// SIMATIC S7-200 project (STEP 7-Micro/WIN), CPU 224 UN REL 02.01

SYMBOL_TABLE 01
数据记录             M0.0     // 0记录 1 不记录
光源模式             M0.1     // 光源模式切换 0新光源 1老光源
设置时钟B            M0.2     // 设置时钟按钮
间隔               M0.3
间隔使能             M0.4
整点               M0.5
在线               M0.6
离线               M0.7
报警复位             M1.0
维护               M1.1
启动标定             M1.2
启动测量             M1.3
自动标定             M1.4
恢复默认             M1.5
无源启动             M1.6
急停               M1.7
运行中              M2.0
实样标记             M3.3
启动质控             M3.4
质控标记             M3.5
质控标定标记           M3.7
量程切换开关           M4.0
加热开关             M5.1
负值显示             M5.2
正常结束             M11.0
连续测试状态           M11.2
历史使能             M20.0
empty            M23.0
进样标记             V19.0
标定中              V20.0
标定阶段0            V20.1
标定阶段1            V20.4
标定阶段2            V21.0
测量中              V22.0
第一档              V91.0
第二档              V91.1
第三档              V91.2
第四档              V91.3
第五档              V91.4
档位               VB90     // 0：第一档  1：第二档  2：第三档  3：第四档
切换范围             VB92
自标时              VB258
自标分              VB259
时钟字节             VB400    // BCD
时钟时              VB403
时钟分              VB404
显色               VD220
基准               VD224
校正系数             VD270
负值区间             VD274
操作密码             VD306
管理密码             VD310
超级密码             VD314
中间值              VD490
模拟输出             VD494
平均电压             VD582
临时A0             VD636
平均A0             VD640
平均A1             VD644
平均A2             VD648
临时A1             VD656
临时A2             VD660
仪器动作             VW94
仪器状态             VW96
占空比              VW218
间隔时              VW230
间隔分              VW232
质不过              VW260
质已测              VW262
切换次数             VW264
标0次数             VW326
标1次数             VW328
标2次数             VW330
HMI窗口号           VW390
时钟字              VW410    // BCD
测量启动时间           VW450
断电时刻             VW470
END_SYMBOL_TABLE

SYMBOL_TABLE 输入输出
下三通信号            I0.0
上三通信号            I0.1
水样浮球             I1.2
废液浮球             I1.3
加热               Q0.0
光源               Q0.1
加热保护             Q0.2
END_SYMBOL_TABLE

SYMBOL_TABLE 自动
A试剂a             V0.0     // 重铬酸钾
B试剂a             V0.1
C试剂a             V0.2     // 硫酸
D试剂a             V0.3
X试剂a             V0.4
纯水a              V0.5
清洗液a             V0.6
水样a              V0.7
空气a              V1.0
进样阀a             V1.1
切水样阀a            V1.2
高压阀a             V1.3
上摇臂a             V1.4
下摇臂a             V1.5
P1抽a             V1.6
P1推a             V1.7
P2抽a             V2.0
P2推a             V2.1
P外a              V2.2
风扇a              V2.3
校一a              V2.4
校二a              V2.5
光源a              V2.6
样校水              V2.7
采样球阀a            V3.0     // 常闭
排空球阀2a           V3.1     // 常开
硫酸a              V3.2
重铬酸钾a            V3.3
备用1a             V3.4
END_SYMBOL_TABLE

SYMBOL_TABLE 参数
校一浓度             VD100    // 浮
校二浓度             VD104    // 浮
消解时间             VW108    // min
显色时间             VW110    // min
采样报警时间           VW112    // min
罐溢流时间            VW114    // s
管溢流时间            VW116    // s
                 VW118    // 测量模式
                 VW120    // 自动标定启用
自标周期             VW122    // 天
当前计算             VW124    // 天
模拟量程             VD126    // mg/L   浮
消解温度             VD130    // 浮
版本号              VD134    // 浮
启动时刻             VW138    // hex   ,vw134-vw142
标定时刻             VW148    // hex    ,vw144-152
K                VD158    // 浮
B                VD162    // 浮
水样A              VD166    // 浮
水样T              VD170    // 浮
校正液T             VD174    // 浮
纯水T              VD178    // 浮
校一A              VD182    // 浮
校二A              VD186    // 浮
当前温度             VD190    // 浮
当前电压             VD194    // 浮
排空电压             VD1100
清洗电压             VD1104
目标温度             VD200
显色温度             VD204
END_SYMBOL_TABLE

SYMBOL_TABLE 报警
A试剂报警            V80.0    // Vb80-81二级报警 ,停止一切操作
B试剂报警            V80.1
C试剂报警            V80.2
D试剂报警            V80.3
X试剂报警            V80.4
纯水报警             V80.5
硫酸报警             V80.6
废液满              V81.0
校一报警             V81.1
校二报警             V81.2
采样报警             V82.1
重铬酸钾报警           V81.4
清洗液报警            V81.5
在线样报警            V82.0    // vb82一级报警，自动测量不停
消解温度异常           V83.0
待机温度异常           V83.1
冷却超时             V83.2
基准偏低             V83.3
END_SYMBOL_TABLE

SYMBOL_TABLE S7-200 符号
Always_On        SM0.0    // 始终接通为 ON
First_Scan_On    SM0.1    // 仅第一个扫描周期中接通为 ON
Clock_1s         SM0.5    // 在 1 秒钟的循环周期内，接通为 ON 0.5 秒，关断为 OFF 0.5  秒
END_SYMBOL_TABLE

ORGANIZATION_BLOCK 程序块:OB1
TITLE=
BEGIN
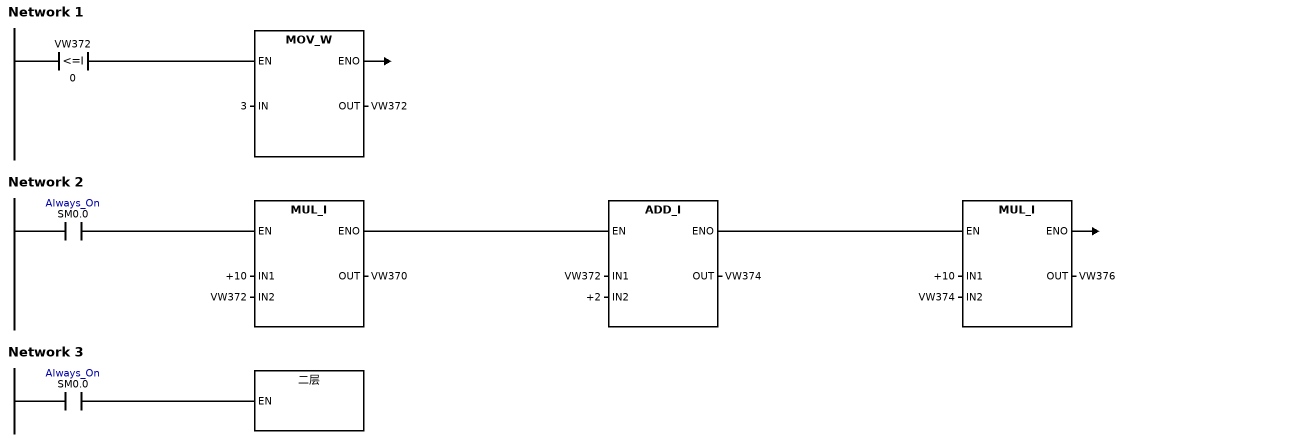
Network 1
LDW<=  VW372, 0
MOVW   3, VW372
Network 2
LD     Always_On:SM0.0
MOVW   +10, VW370
AENO
*I     VW372, VW370
AENO
MOVW   VW372, VW374
AENO
+I     +2, VW374
AENO
MOVW   +10, VW376
*I     VW374, VW376
Network 3
LD     Always_On:SM0.0
CALL   二层:SBR10
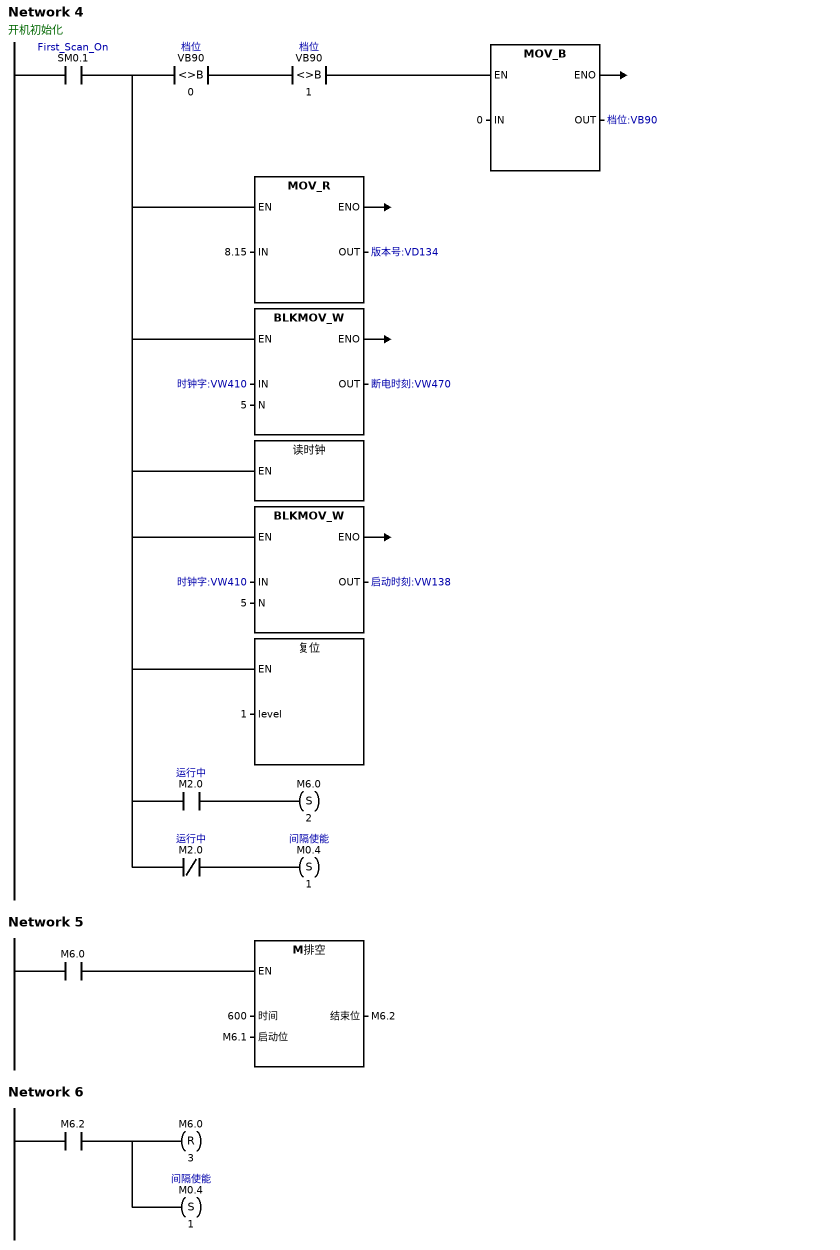
Network 4
// 开机初始化
LD     First_Scan_On:SM0.1
LPS
AB<>   档位:VB90, 0
AB<>   档位:VB90, 1
MOVB   0, 档位:VB90
LRD
MOVR   8.15, 版本号:VD134
LRD
BMW    时钟字:VW410, 断电时刻:VW470, 5
LRD
CALL   读时钟:SBR28
LRD
BMW    时钟字:VW410, 启动时刻:VW138, 5
LRD
CALL   复位:SBR34, 1
LRD
A      运行中:M2.0
S      M6.0, 2
LPP
AN     运行中:M2.0
S      间隔使能:M0.4, 1
Network 5
LD     M6.0
CALL   M排空:SBR5, 600, M6.1, M6.2
Network 6
LD     M6.2
R      M6.0, 3
S      间隔使能:M0.4, 1
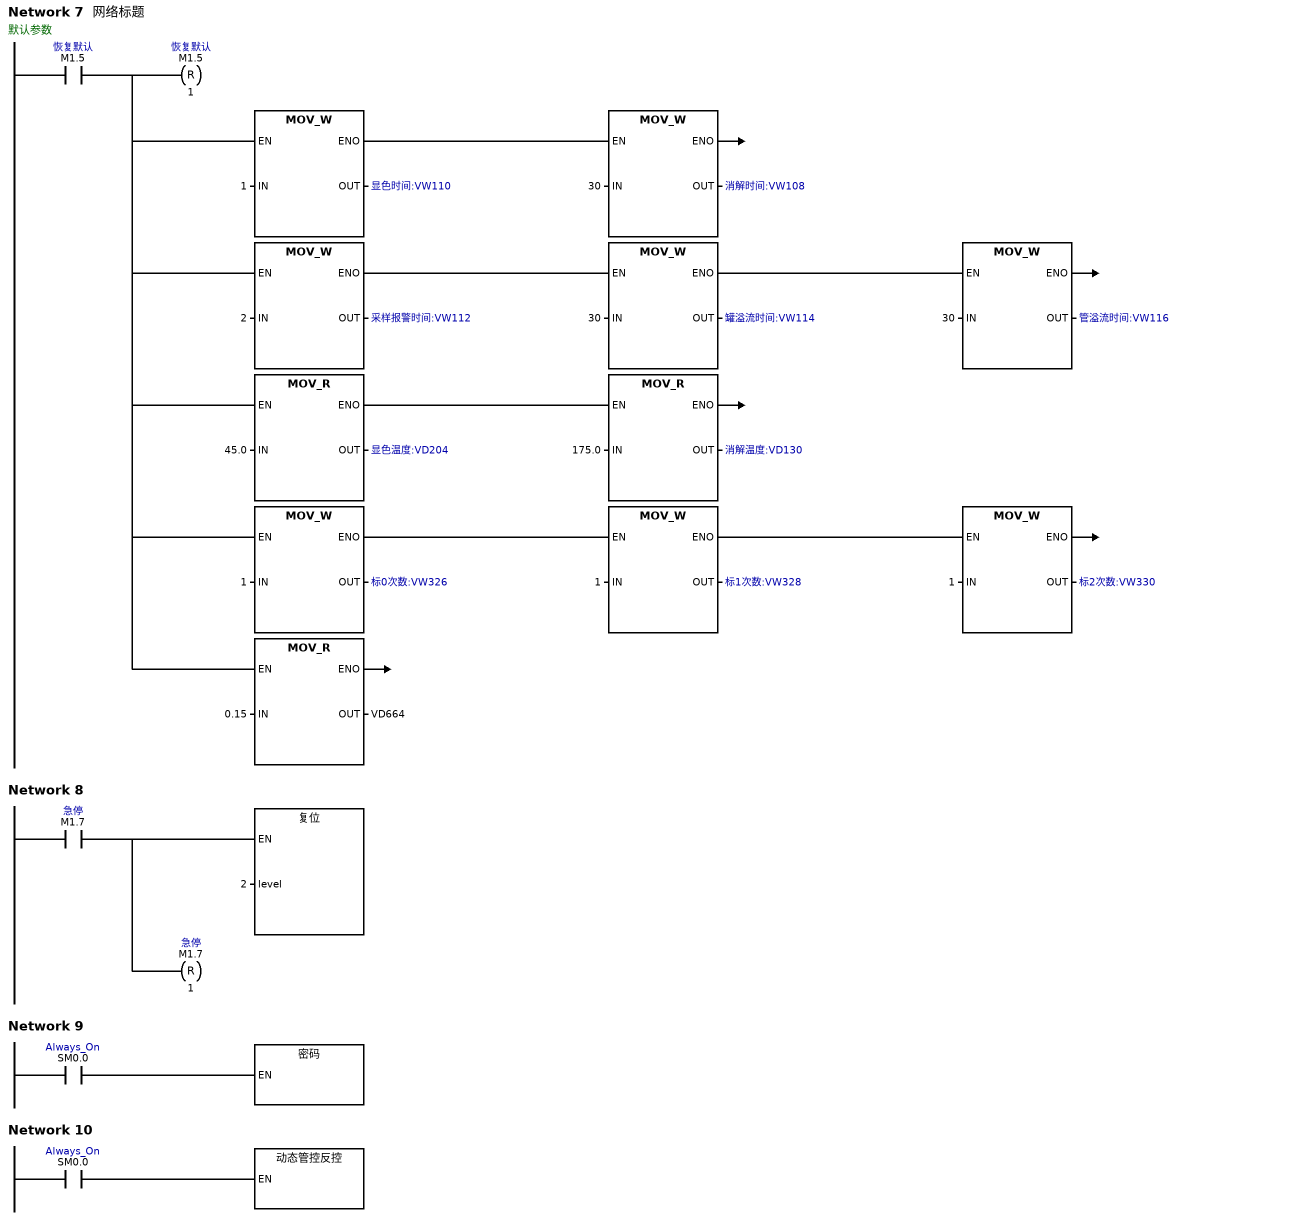
Network 7 // 网络标题
// 默认参数
LD     恢复默认:M1.5
LPS
R      恢复默认:M1.5, 1
MOVW   1, 显色时间:VW110
AENO
MOVW   30, 消解时间:VW108
LRD
MOVW   2, 采样报警时间:VW112
AENO
MOVW   30, 罐溢流时间:VW114
AENO
MOVW   30, 管溢流时间:VW116
LRD
MOVR   45.0, 显色温度:VD204
AENO
MOVR   175.0, 消解温度:VD130
LRD
MOVW   1, 标0次数:VW326
AENO
MOVW   1, 标1次数:VW328
AENO
MOVW   1, 标2次数:VW330
LPP
MOVR   0.15, VD664
Network 8
LD     急停:M1.7
CALL   复位:SBR34, 2
R      急停:M1.7, 1
Network 9
LD     Always_On:SM0.0
CALL   密码:SBR26
Network 10
LD     Always_On:SM0.0
CALL   动态管控反控:SBR38
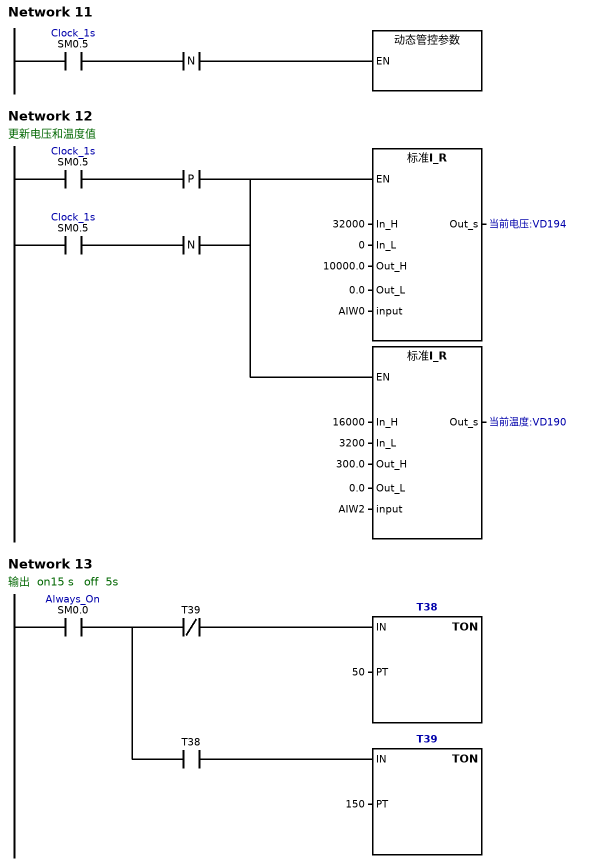
Network 11
LD     Clock_1s:SM0.5
ED
CALL   动态管控参数:SBR24
Network 12
// 更新电压和温度值
LD     Clock_1s:SM0.5
EU
LD     Clock_1s:SM0.5
ED
OLD
CALL   标准I_R:SBR2, 32000, 0, 10000.0, 0.0, AIW0, 当前电压:VD194
CALL   标准I_R:SBR2, 16000, 3200, 300.0, 0.0, AIW2, 当前温度:VD190
Network 13
// 输出  on15 s   off  5s
LD     Always_On:SM0.0
LPS
AN     T39
TON    T38, 50
LPP
A      T38
TON    T39, 150
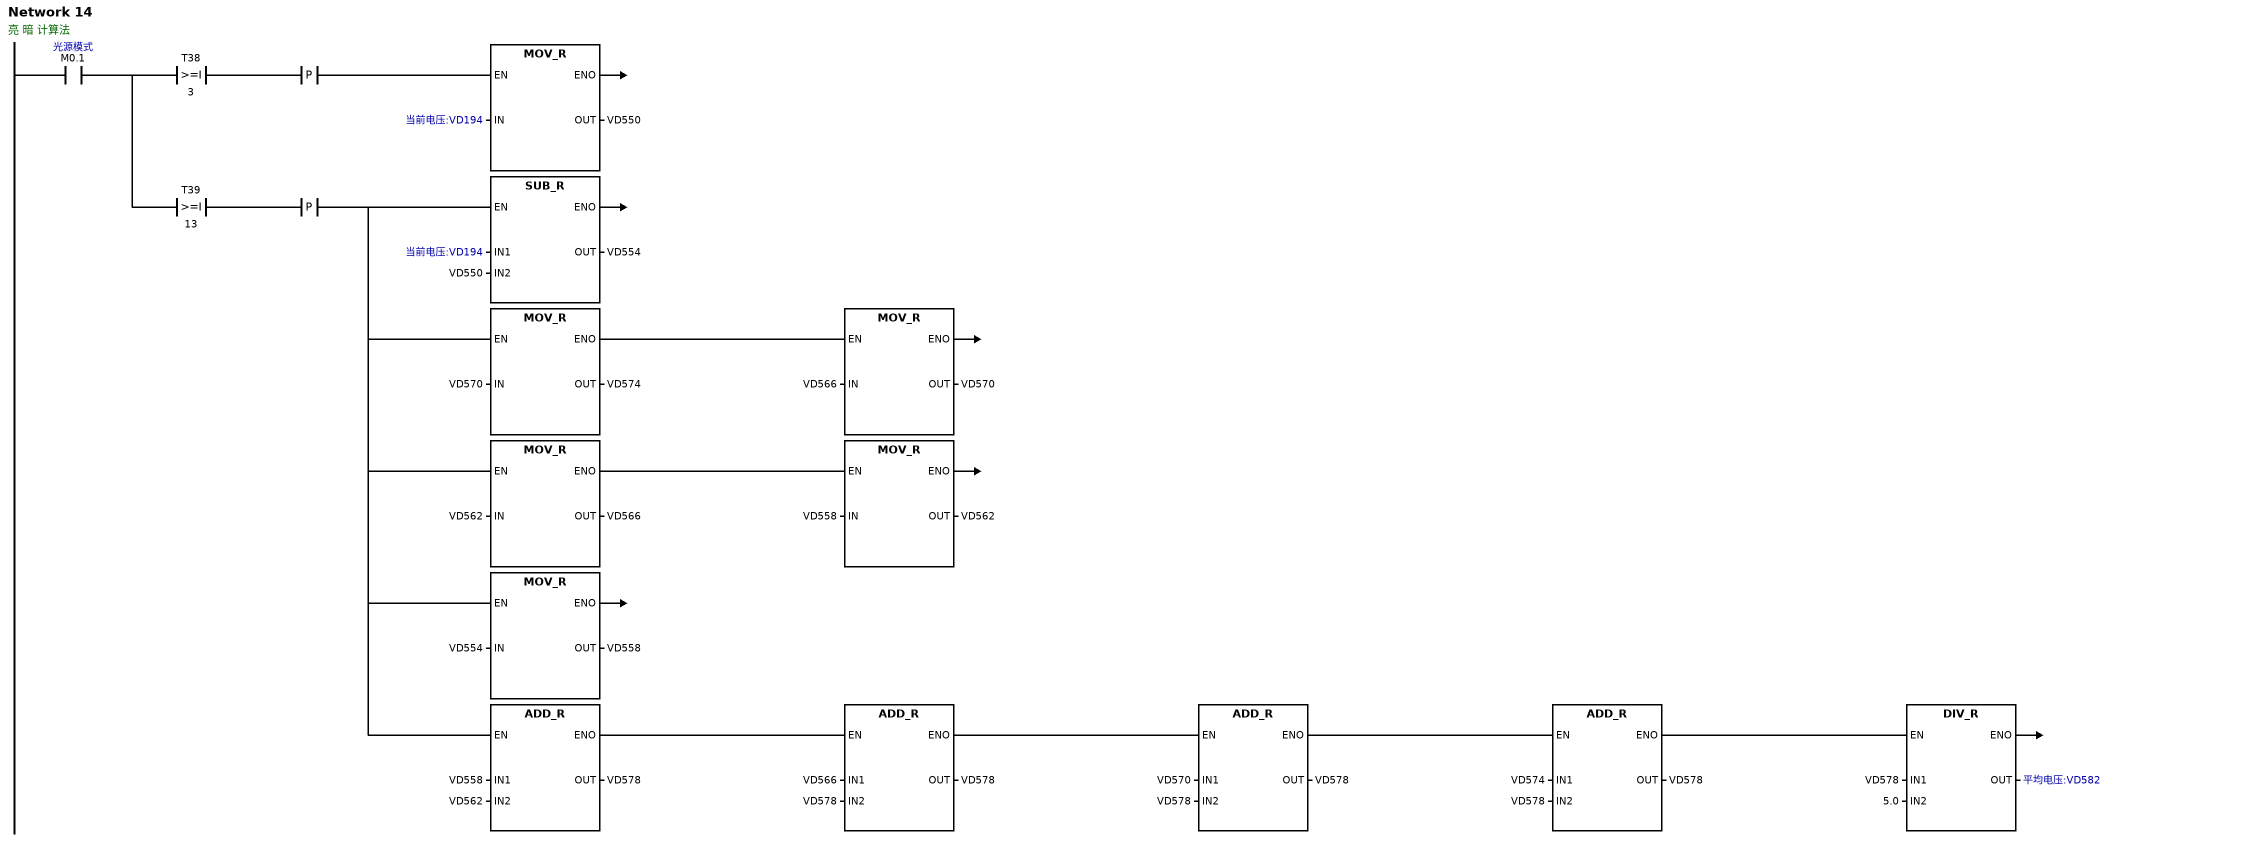
Network 14
// 亮 暗 计算法
LD     光源模式:M0.1
LPS
AW>=   T38, 3
EU
MOVR   当前电压:VD194, VD550
LPP
AW>=   T39, 13
EU
LPS
MOVR   当前电压:VD194, VD554
-R     VD550, VD554
MOVR   VD570, VD574
AENO
MOVR   VD566, VD570
LRD
MOVR   VD562, VD566
AENO
MOVR   VD558, VD562
LRD
MOVR   VD554, VD558
LPP
MOVR   VD558, VD578
AENO
+R     VD562, VD578
AENO
+R     VD566, VD578
AENO
+R     VD570, VD578
AENO
+R     VD574, VD578
AENO
MOVR   VD578, 平均电压:VD582
/R     5.0, 平均电压:VD582
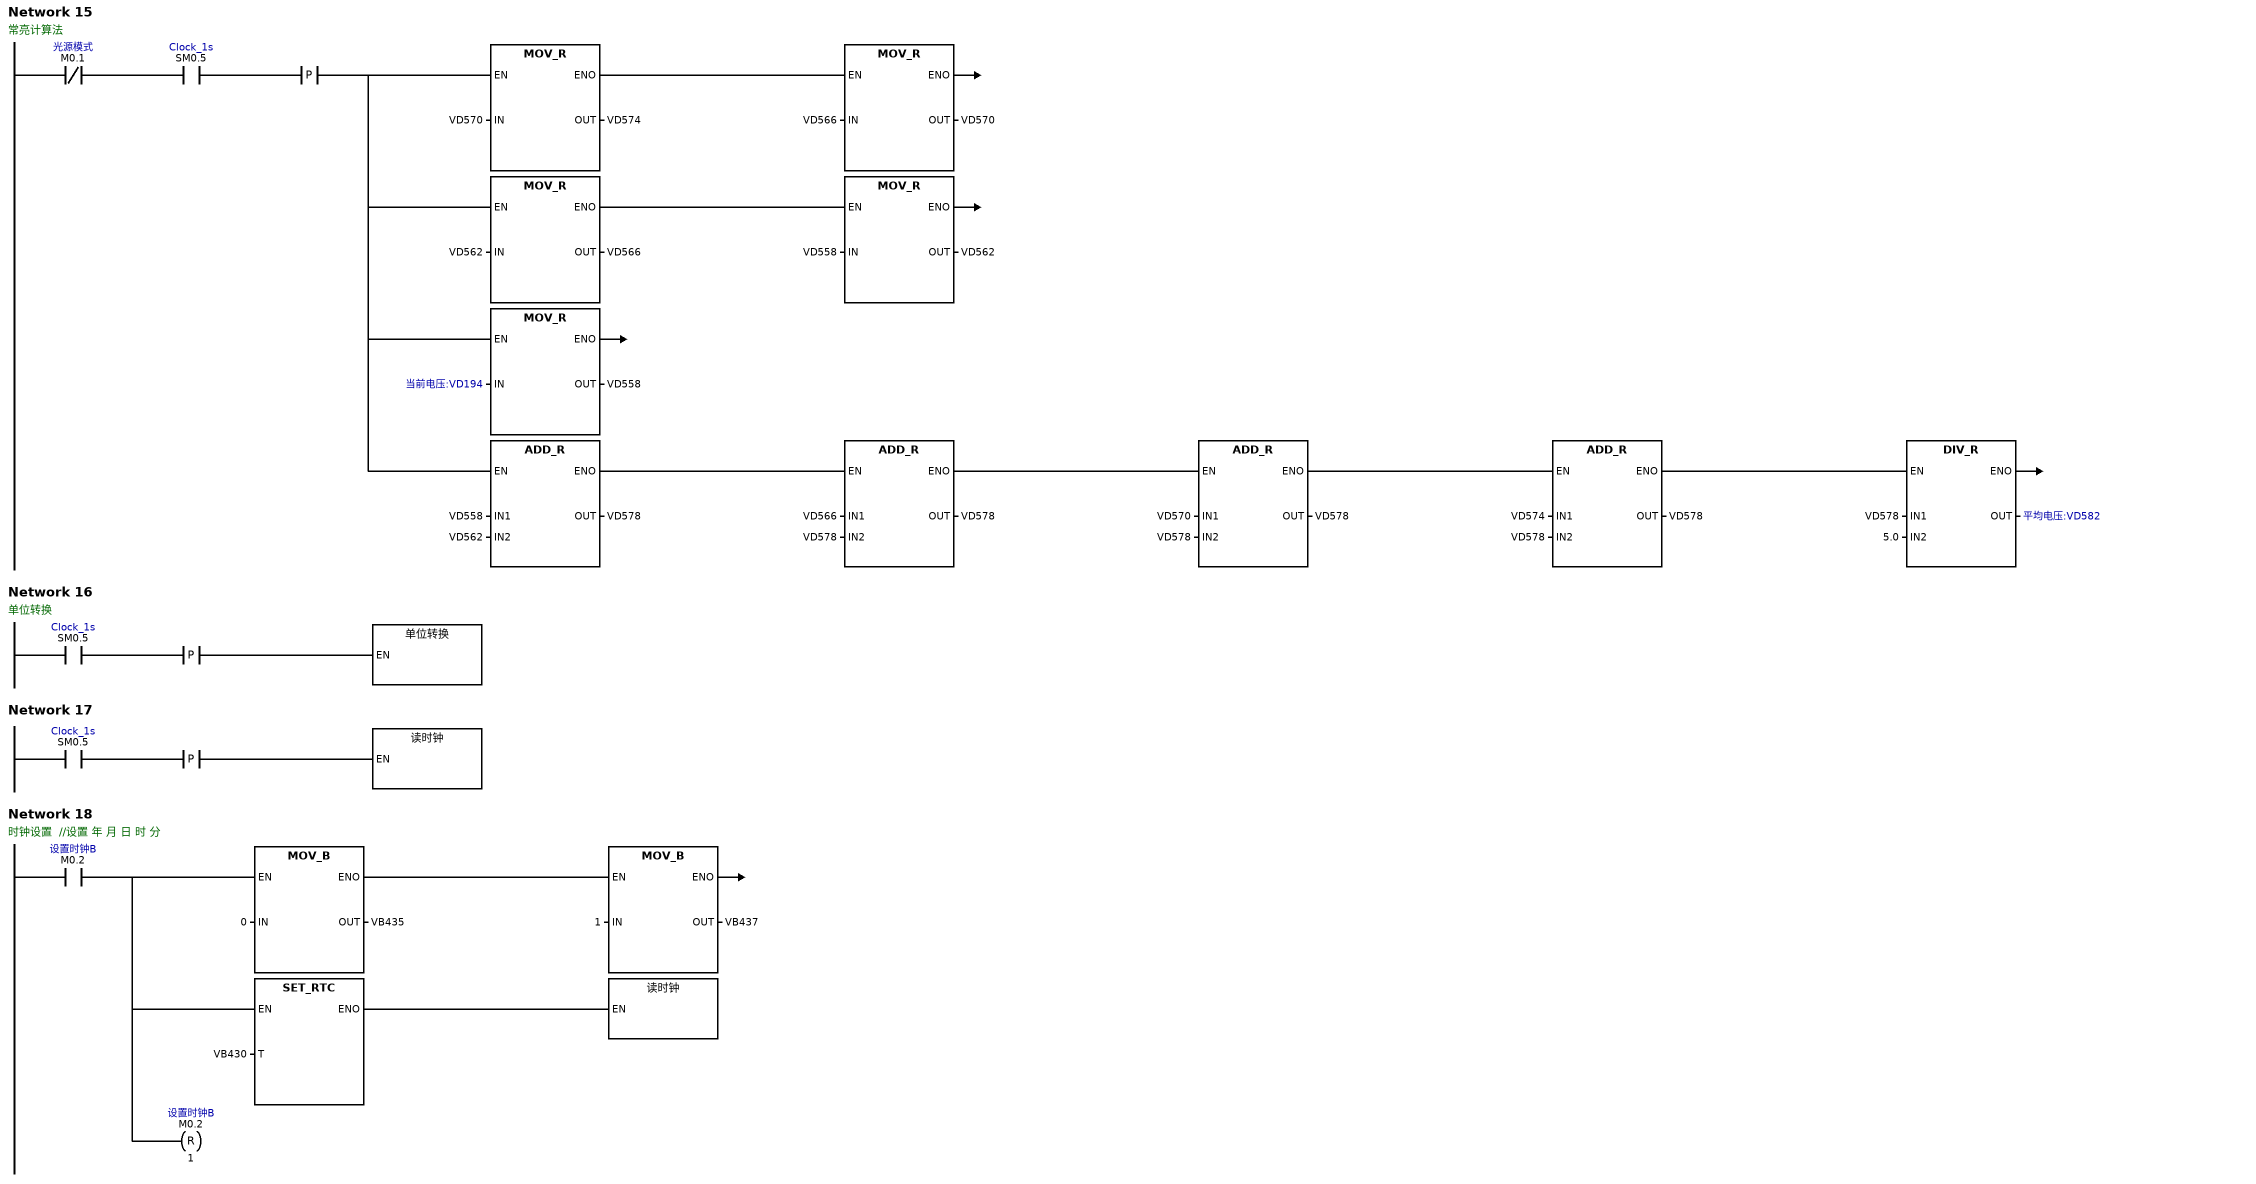
Network 15
// 常亮计算法
LDN    光源模式:M0.1
A      Clock_1s:SM0.5
EU
LPS
MOVR   VD570, VD574
AENO
MOVR   VD566, VD570
LRD
MOVR   VD562, VD566
AENO
MOVR   VD558, VD562
LRD
MOVR   当前电压:VD194, VD558
LPP
MOVR   VD558, VD578
AENO
+R     VD562, VD578
AENO
+R     VD566, VD578
AENO
+R     VD570, VD578
AENO
+R     VD574, VD578
AENO
MOVR   VD578, 平均电压:VD582
/R     5.0, 平均电压:VD582
Network 16
// 单位转换
LD     Clock_1s:SM0.5
EU
CALL   单位转换:SBR27
Network 17
LD     Clock_1s:SM0.5
EU
CALL   读时钟:SBR28
Network 18
// 时钟设置  //设置 年 月 日 时 分
LD     设置时钟B:M0.2
LPS
MOVB   0, VB435
AENO
MOVB   1, VB437
LRD
TODW   VB430
AENO
CALL   读时钟:SBR28
LPP
R      设置时钟B:M0.2, 1
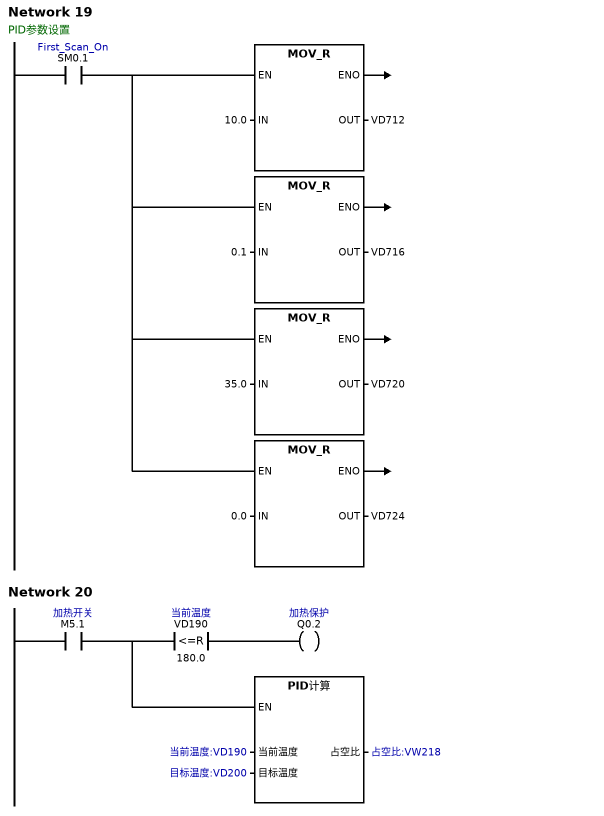
Network 19
// PID参数设置
LD     First_Scan_On:SM0.1
MOVR   10.0, VD712
MOVR   0.1, VD716
MOVR   35.0, VD720
MOVR   0.0, VD724
Network 20
LD     加热开关:M5.1
LPS
AR<=   当前温度:VD190, 180.0
=      加热保护:Q0.2
LPP
CALL   PID计算:SBR9, 当前温度:VD190, 目标温度:VD200, 占空比:VW218
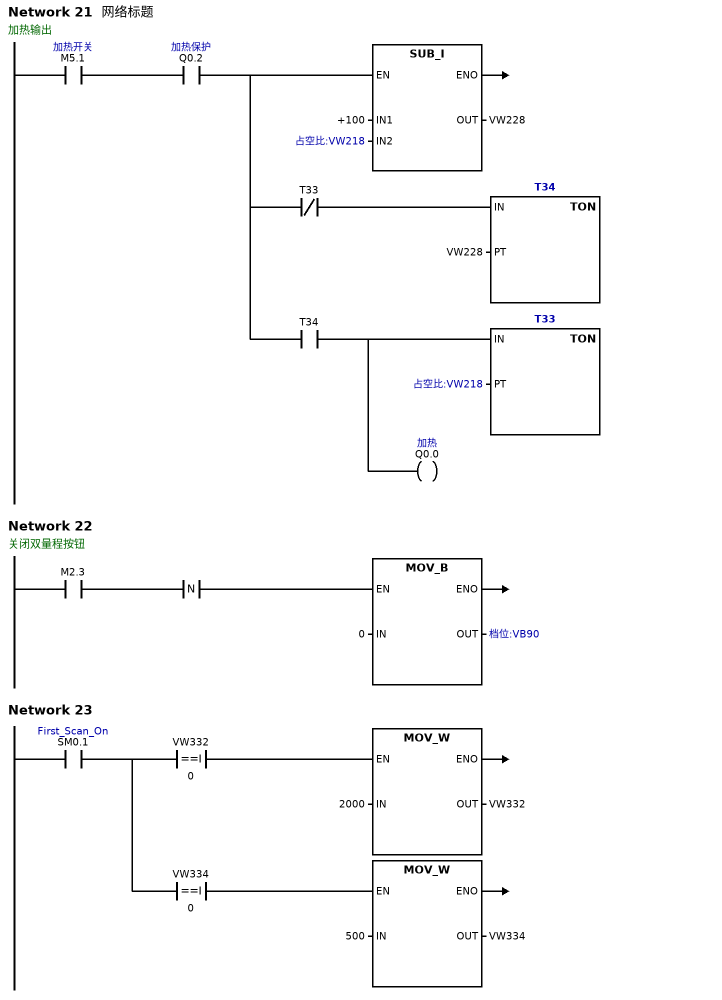
Network 21 // 网络标题
//   加热输出
LD     加热开关:M5.1
A      加热保护:Q0.2
LPS
MOVW   +100, VW228
-I     占空比:VW218, VW228
AN     T33
TON    T34, VW228
LPP
A      T34
TON    T33, 占空比:VW218
=      加热:Q0.0
Network 22
// 关闭双量程按钮
LD     M2.3
ED
MOVB   0, 档位:VB90
Network 23
LD     First_Scan_On:SM0.1
LPS
AW=    VW332, 0
MOVW   2000, VW332
LPP
AW=    VW334, 0
MOVW   500, VW334
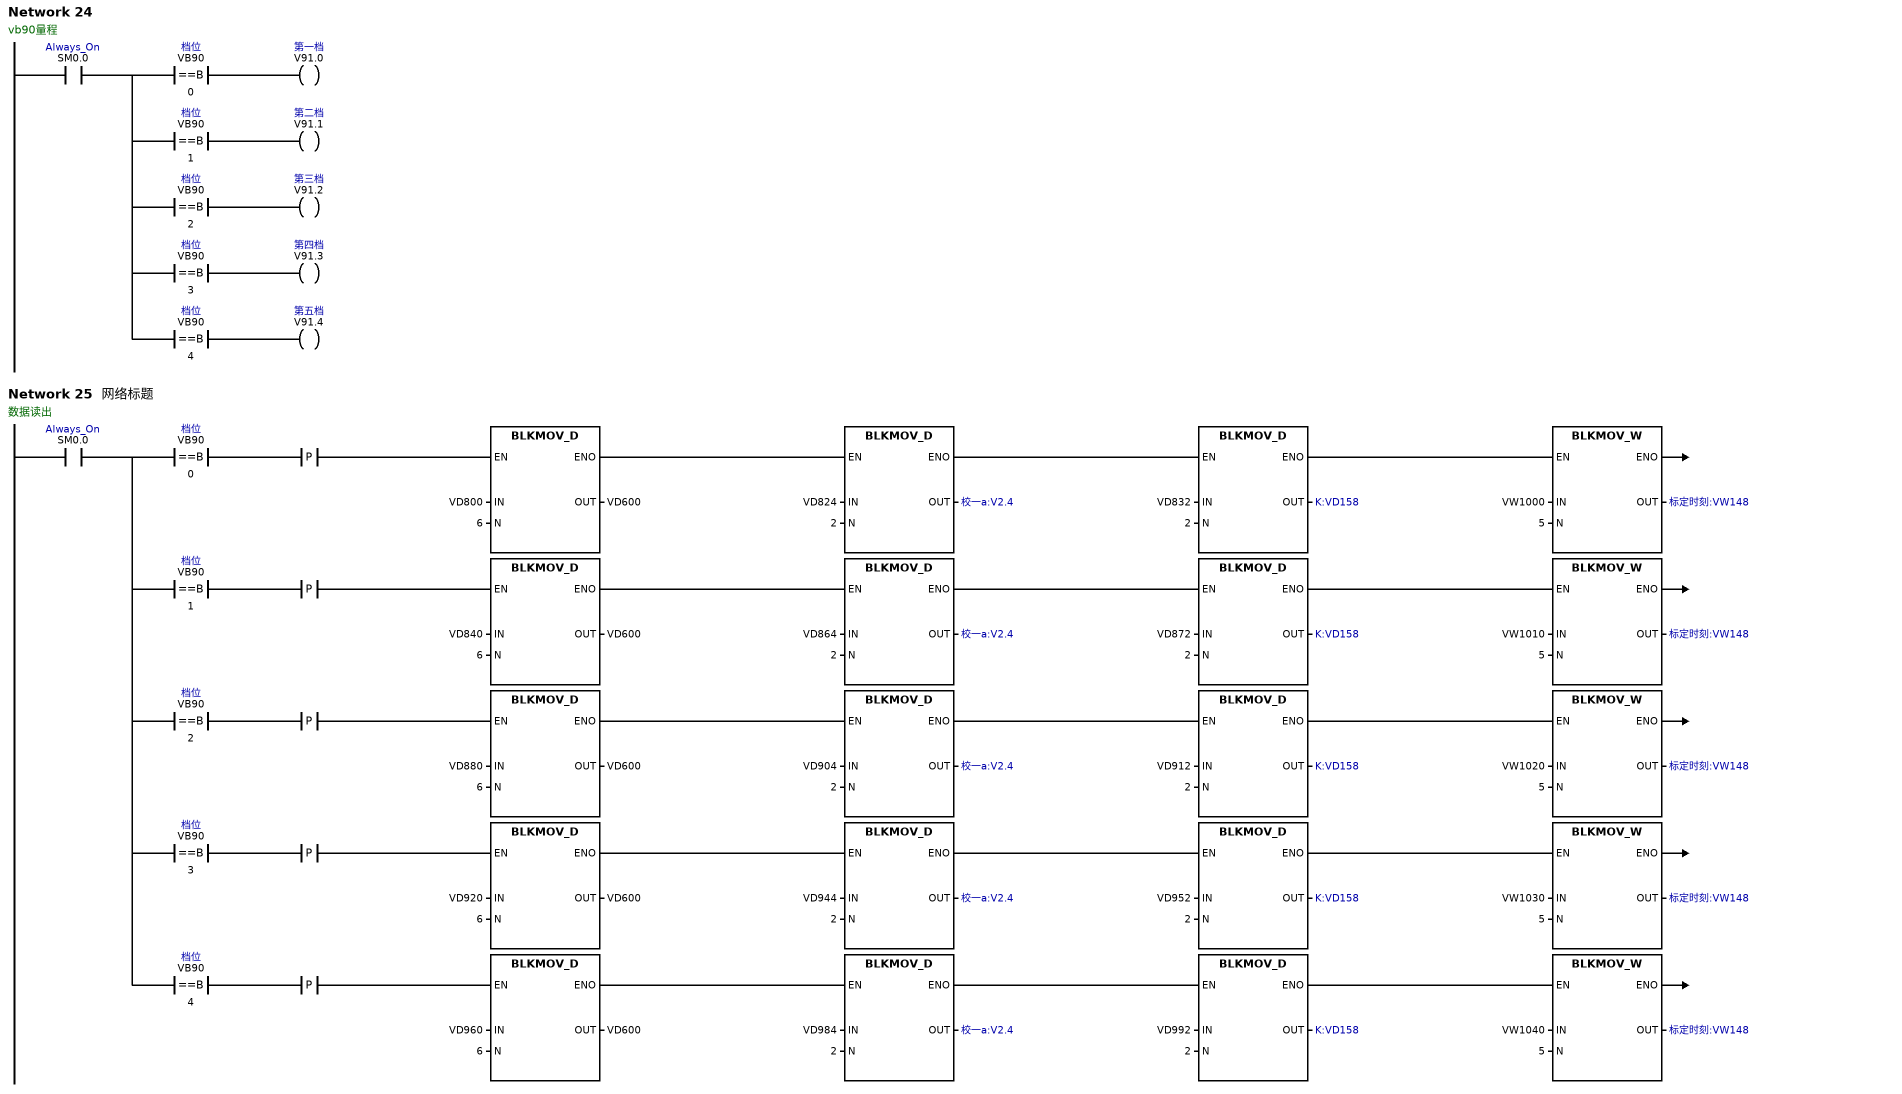
Network 24
// vb90量程
LD     Always_On:SM0.0
LPS
AB=    档位:VB90, 0
=      第一档:V91.0
LRD
AB=    档位:VB90, 1
=      第二档:V91.1
LRD
AB=    档位:VB90, 2
=      第三档:V91.2
LRD
AB=    档位:VB90, 3
=      第四档:V91.3
LPP
AB=    档位:VB90, 4
=      第五档:V91.4
Network 25 // 网络标题
// 数据读出
// (network saved uncompiled; LAD cells follow)
// row 0: c0 -| |- Always_On:SM0.0 v  c1 -|==B|- 档位:VB90, 0  c2 -|P|-  c3 --  c4 [BLKMOV_D EN:=power@row0, IN:=VD800, N:=6, ENO=>power, OUT=>VD600]  c5 --  c6 --  c7 [BLKMOV_D EN:=power@row0, IN:=VD824, N:=2, ENO=>power, OUT=>校一a:V2.4]  c8 --  c9 --  c10 [BLKMOV_D EN:=power@row0, IN:=VD832, N:=2, ENO=>power, OUT=>K:VD158]  c11 --  c12 --  c13 [BLKMOV_W EN:=power@row0, IN:=VW1000, N:=5, ENO=>power, OUT=>标定时刻:VW148]  c14 ->
// row 1: c0 ^v  c4 [box]  c7 [box]  c10 [box]  c13 [box]
// row 2: c0 ^v  c1 -|==B|- 档位:VB90, 1  c2 -|P|-  c3 --  c4 [BLKMOV_D EN:=power@row2, IN:=VD840, N:=6, ENO=>power, OUT=>VD600]  c5 --  c6 --  c7 [BLKMOV_D EN:=power@row2, IN:=VD864, N:=2, ENO=>power, OUT=>校一a:V2.4]  c8 --  c9 --  c10 [BLKMOV_D EN:=power@row2, IN:=VD872, N:=2, ENO=>power, OUT=>K:VD158]  c11 --  c12 --  c13 [BLKMOV_W EN:=power@row2, IN:=VW1010, N:=5, ENO=>power, OUT=>标定时刻:VW148]  c14 ->
// row 3: c0 ^v  c4 [box]  c7 [box]  c10 [box]  c13 [box]
// row 4: c0 ^v  c1 -|==B|- 档位:VB90, 2  c2 -|P|-  c3 --  c4 [BLKMOV_D EN:=power@row4, IN:=VD880, N:=6, ENO=>power, OUT=>VD600]  c5 --  c6 --  c7 [BLKMOV_D EN:=power@row4, IN:=VD904, N:=2, ENO=>power, OUT=>校一a:V2.4]  c8 --  c9 --  c10 [BLKMOV_D EN:=power@row4, IN:=VD912, N:=2, ENO=>power, OUT=>K:VD158]  c11 --  c12 --  c13 [BLKMOV_W EN:=power@row4, IN:=VW1020, N:=5, ENO=>power, OUT=>标定时刻:VW148]  c14 ->
// row 5: c0 ^v  c4 [box]  c7 [box]  c10 [box]  c13 [box]
// row 6: c0 ^v  c1 -|==B|- 档位:VB90, 3  c2 -|P|-  c3 --  c4 [BLKMOV_D EN:=power@row6, IN:=VD920, N:=6, ENO=>power, OUT=>VD600]  c5 --  c6 --  c7 [BLKMOV_D EN:=power@row6, IN:=VD944, N:=2, ENO=>power, OUT=>校一a:V2.4]  c8 --  c9 --  c10 [BLKMOV_D EN:=power@row6, IN:=VD952, N:=2, ENO=>power, OUT=>K:VD158]  c11 --  c12 --  c13 [BLKMOV_W EN:=power@row6, IN:=VW1030, N:=5, ENO=>power, OUT=>标定时刻:VW148]  c14 ->
// row 7: c0 ^v  c4 [box]  c7 [box]  c10 [box]  c13 [box]
// row 8: c0 ^  c1 -|==B|- 档位:VB90, 4  c2 -|P|-  c3 --  c4 [BLKMOV_D EN:=power@row8, IN:=VD960, N:=6, ENO=>power, OUT=>VD600]  c5 --  c6 --  c7 [BLKMOV_D EN:=power@row8, IN:=VD984, N:=2, ENO=>power, OUT=>校一a:V2.4]  c8 --  c9 --  c10 [BLKMOV_D EN:=power@row8, IN:=VD992, N:=2, ENO=>power, OUT=>K:VD158]  c11 --  c12 --  c13 [BLKMOV_W EN:=power@row8, IN:=VW1040, N:=5, ENO=>power, OUT=>标定时刻:VW148]  c14 ->
// row 9: c4 [box]  c7 [box]  c10 [box]  c13 [box]
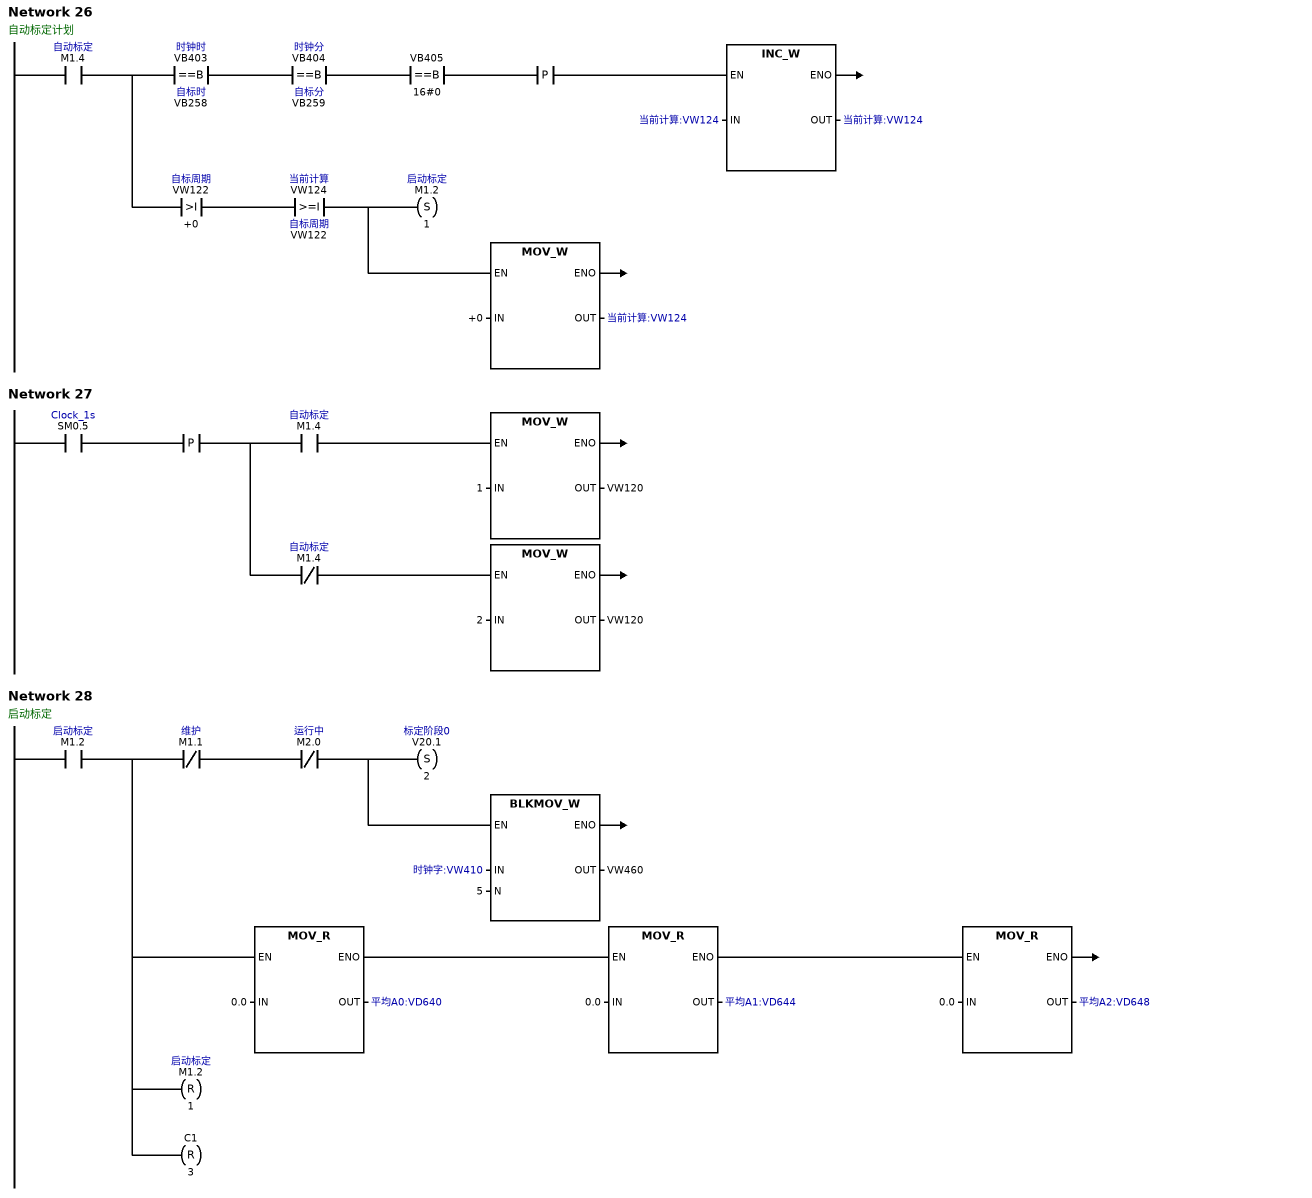
Network 26
// 自动标定计划
LD     自动标定:M1.4
LPS
AB=    时钟时:VB403, 自标时:VB258
AB=    时钟分:VB404, 自标分:VB259
AB=    VB405, 16#0
EU
INCW   当前计算:VW124
LPP
AW>    自标周期:VW122, +0
AW>=   当前计算:VW124, 自标周期:VW122
S      启动标定:M1.2, 1
MOVW   +0, 当前计算:VW124
Network 27
LD     Clock_1s:SM0.5
EU
LPS
A      自动标定:M1.4
MOVW   1, VW120
LPP
AN     自动标定:M1.4
MOVW   2, VW120
Network 28
// 启动标定
LD     启动标定:M1.2
LPS
AN     维护:M1.1
AN     运行中:M2.0
S      标定阶段0:V20.1, 2
BMW    时钟字:VW410, VW460, 5
LPP
LPS
MOVR   0.0, 平均A0:VD640
AENO
MOVR   0.0, 平均A1:VD644
AENO
MOVR   0.0, 平均A2:VD648
LRD
R      启动标定:M1.2, 1
LPP
R      C1, 3
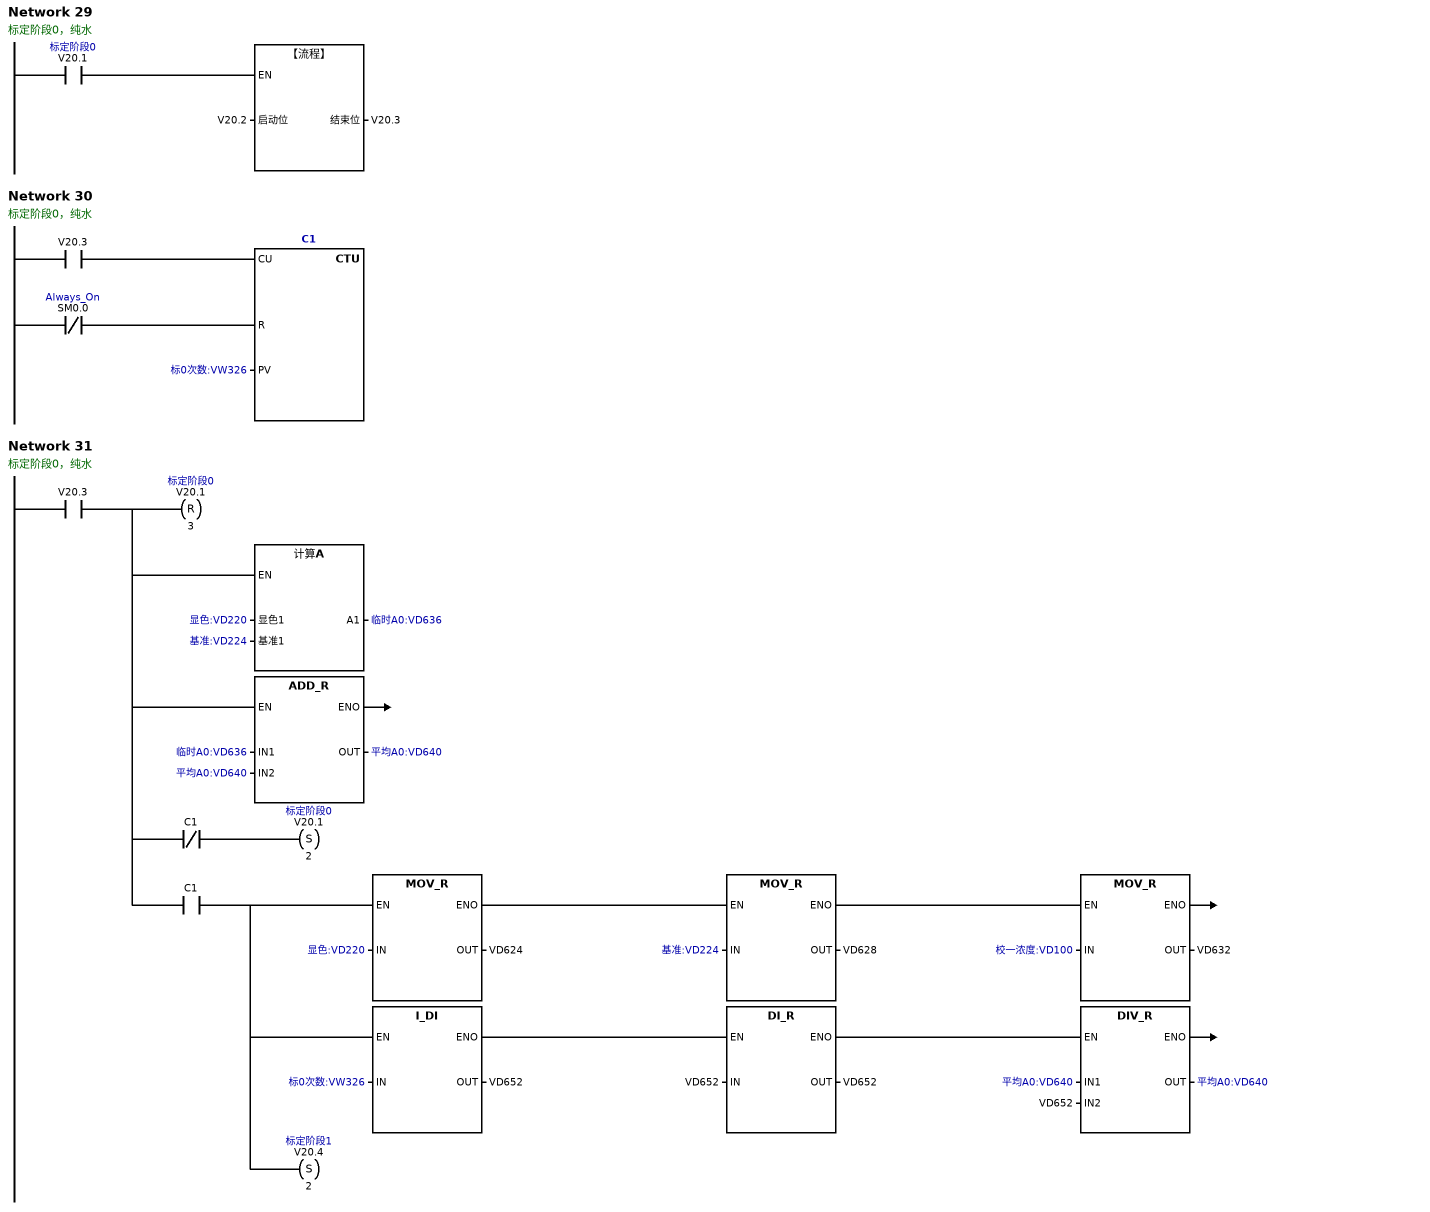
Network 29
// 标定阶段0，纯水
LD     标定阶段0:V20.1
CALL   【流程】:SBR7, V20.2, V20.3
Network 30
// 标定阶段0，纯水
LD     V20.3
LDN    Always_On:SM0.0
CTU    C1, 标0次数:VW326
Network 31
// 标定阶段0，纯水
LD     V20.3
LPS
R      标定阶段0:V20.1, 3
CALL   计算A:SBR37, 显色:VD220, 基准:VD224, 临时A0:VD636
+R     临时A0:VD636, 平均A0:VD640
AN     C1
S      标定阶段0:V20.1, 2
LPP
A      C1
LPS
MOVR   显色:VD220, VD624
AENO
MOVR   基准:VD224, VD628
AENO
MOVR   校一浓度:VD100, VD632
LRD
ITD    标0次数:VW326, VD652
AENO
DTR    VD652, VD652
AENO
/R     VD652, 平均A0:VD640
LPP
S      标定阶段1:V20.4, 2
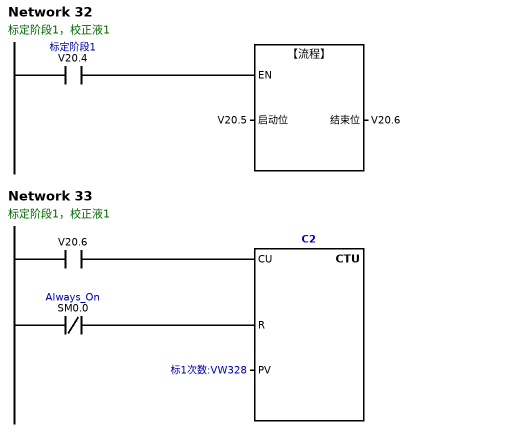
Network 32
// 标定阶段1，校正液1
LD     标定阶段1:V20.4
CALL   【流程】:SBR7, V20.5, V20.6
Network 33
// 标定阶段1，校正液1
LD     V20.6
LDN    Always_On:SM0.0
CTU    C2, 标1次数:VW328
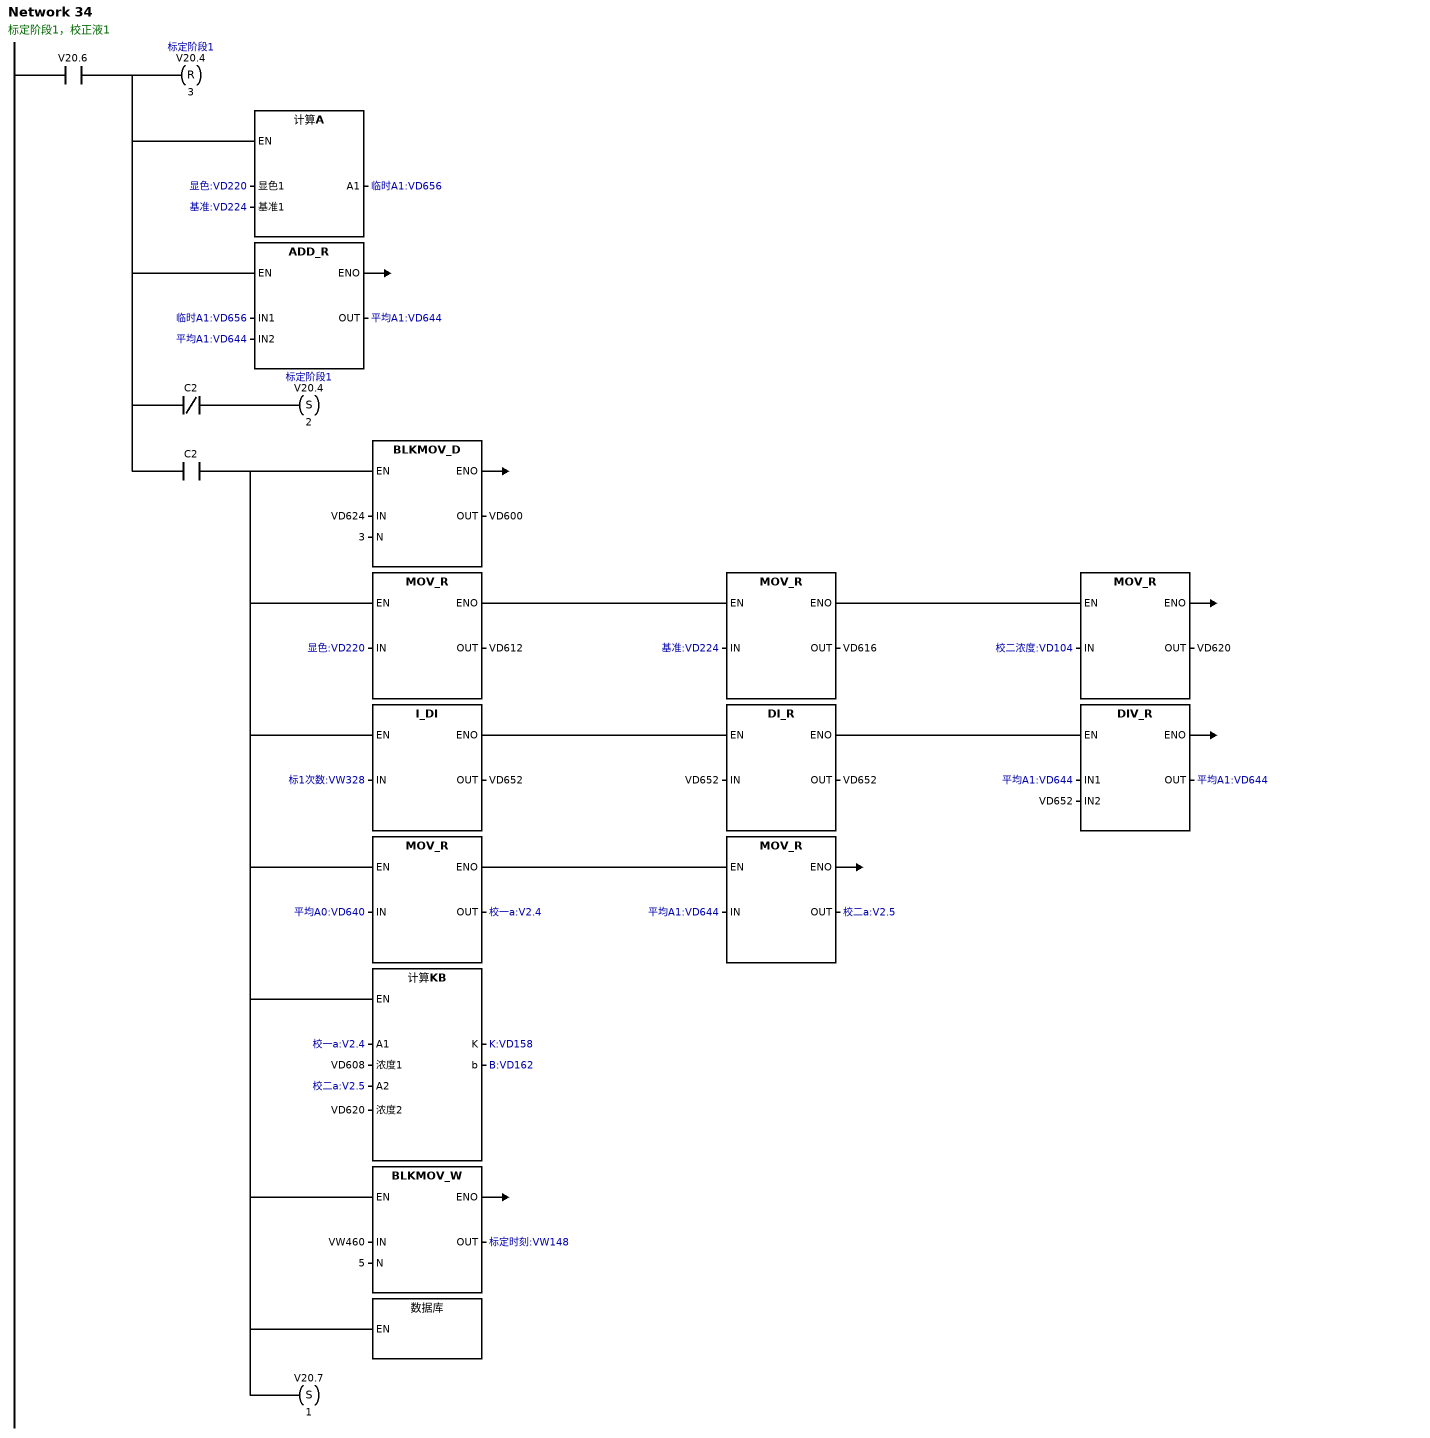
Network 34
// 标定阶段1，校正液1
// (network saved uncompiled; LAD cells follow)
// row 0: c0 -| |- V20.6 v  c1 -(R) 标定阶段1:V20.4, 3
// row 1: c0 ^v  c1 --  c2 [计算A EN:=power@row1, 显色1:=显色:VD220, 基准1:=基准:VD224, A1=>临时A1:VD656]
// row 2: c0 ^v  c2 [box]
// row 3: c0 ^v  c1 --  c2 [ADD_R EN:=power@row3, IN1:=临时A1:VD656, IN2:=平均A1:VD644, ENO=>power, OUT=>平均A1:VD644]  c3 ->
// row 4: c0 ^v  c2 [box]
// row 5: c0 ^v  c1 -|/|- C2  c2 -(S) 标定阶段1:V20.4, 2
// row 6: c0 ^  c1 -| |- C2 v  c2 --  c3 [BLKMOV_D EN:=power@row6, IN:=VD624, N:=3, ENO=>power, OUT=>VD600]  c4 ->
// row 7: c1 ^v  c3 [box]
// row 8: c1 ^v  c2 --  c3 [MOV_R EN:=power@row8, IN:=显色:VD220, ENO=>power, OUT=>VD612]  c4 --  c5 --  c6 [MOV_R EN:=power@row8, IN:=基准:VD224, ENO=>power, OUT=>VD616]  c7 --  c8 --  c9 [MOV_R EN:=power@row8, IN:=校二浓度:VD104, ENO=>power, OUT=>VD620]  c10 ->
// row 9: c1 ^v  c3 [box]  c6 [box]  c9 [box]
// row 10: c1 ^v  c2 --  c3 [I_DI EN:=power@row10, IN:=标1次数:VW328, ENO=>power, OUT=>VD652]  c4 --  c5 --  c6 [DI_R EN:=power@row10, IN:=VD652, ENO=>power, OUT=>VD652]  c7 --  c8 --  c9 [DIV_R EN:=power@row10, IN1:=平均A1:VD644, IN2:=VD652, ENO=>power, OUT=>平均A1:VD644]  c10 ->
// row 11: c1 ^v  c3 [box]  c6 [box]  c9 [box]
// row 12: c1 ^v  c2 --  c3 [MOV_R EN:=power@row12, IN:=平均A0:VD640, ENO=>power, OUT=>校一a:V2.4]  c4 --  c5 --  c6 [MOV_R EN:=power@row12, IN:=平均A1:VD644, ENO=>power, OUT=>校二a:V2.5]  c7 ->
// row 13: c1 ^v  c3 [box]  c6 [box]
// row 14: c1 ^v  c2 --  c3 [计算KB EN:=power@row14, A1:=校一a:V2.4, 浓度1:=VD608, A2:=校二a:V2.5, 浓度2:=VD620, K=>K:VD158, b=>B:VD162]
// row 15: c1 ^v  c3 [box]
// row 16: c1 ^v  c3 [box]
// row 17: c1 ^v  c2 --  c3 [BLKMOV_W EN:=power@row17, IN:=VW460, N:=5, ENO=>power, OUT=>标定时刻:VW148]  c4 ->
// row 18: c1 ^v  c3 [box]
// row 19: c1 ^v  c2 --  c3 [数据库 EN:=power@row19]
// row 20: c1 ^  c2 -(S) V20.7, 1
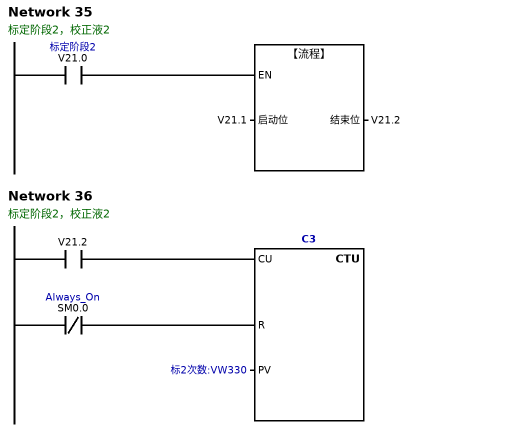
Network 35
// 标定阶段2，校正液2
LD     标定阶段2:V21.0
CALL   【流程】:SBR7, V21.1, V21.2
Network 36
// 标定阶段2，校正液2
LD     V21.2
LDN    Always_On:SM0.0
CTU    C3, 标2次数:VW330
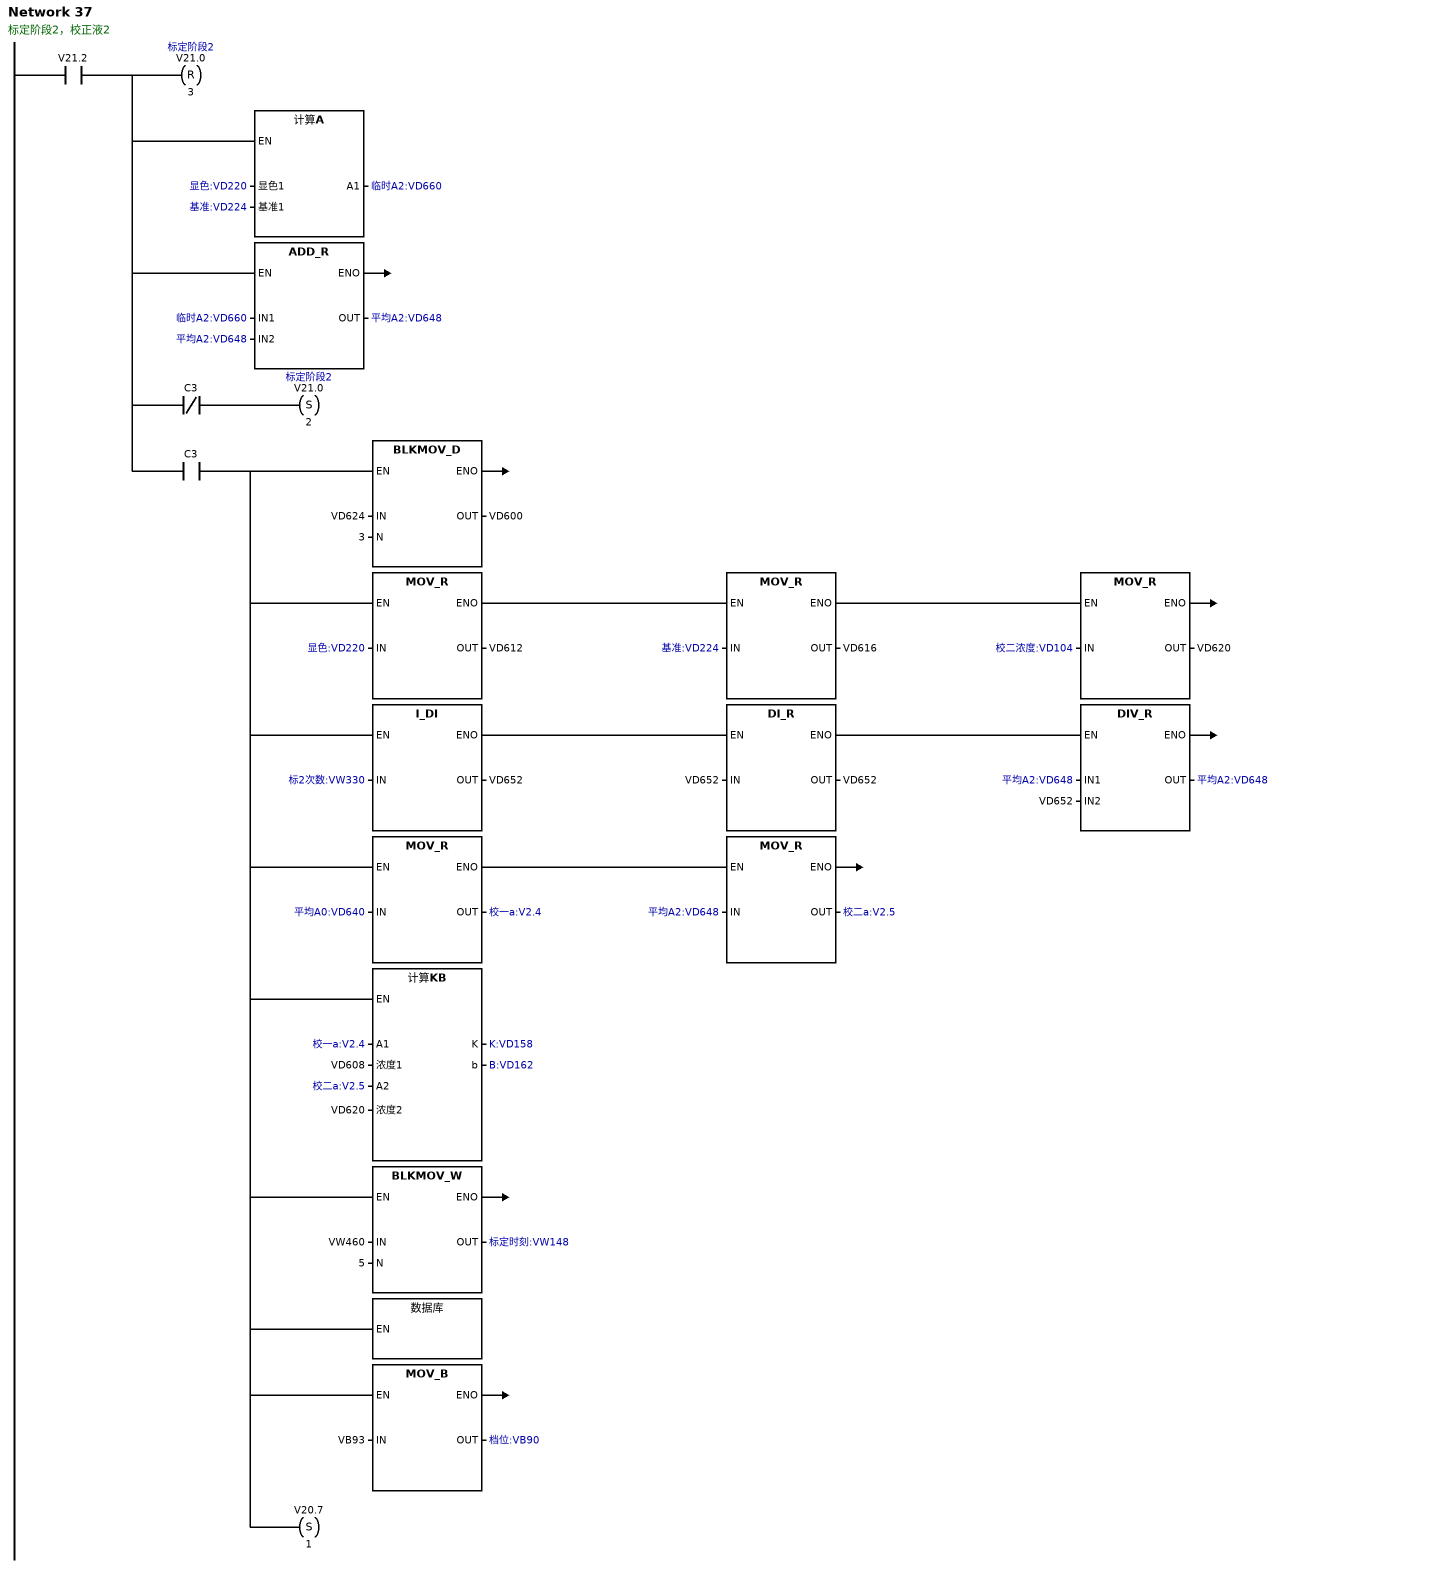
Network 37
// 标定阶段2，校正液2
// (network saved uncompiled; LAD cells follow)
// row 0: c0 -| |- V21.2 v  c1 -(R) 标定阶段2:V21.0, 3
// row 1: c0 ^v  c1 --  c2 [计算A EN:=power@row1, 显色1:=显色:VD220, 基准1:=基准:VD224, A1=>临时A2:VD660]
// row 2: c0 ^v  c2 [box]
// row 3: c0 ^v  c1 --  c2 [ADD_R EN:=power@row3, IN1:=临时A2:VD660, IN2:=平均A2:VD648, ENO=>power, OUT=>平均A2:VD648]  c3 ->
// row 4: c0 ^v  c2 [box]
// row 5: c0 ^v  c1 -|/|- C3  c2 -(S) 标定阶段2:V21.0, 2
// row 6: c0 ^  c1 -| |- C3 v  c2 --  c3 [BLKMOV_D EN:=power@row6, IN:=VD624, N:=3, ENO=>power, OUT=>VD600]  c4 ->
// row 7: c1 ^v  c3 [box]
// row 8: c1 ^v  c2 --  c3 [MOV_R EN:=power@row8, IN:=显色:VD220, ENO=>power, OUT=>VD612]  c4 --  c5 --  c6 [MOV_R EN:=power@row8, IN:=基准:VD224, ENO=>power, OUT=>VD616]  c7 --  c8 --  c9 [MOV_R EN:=power@row8, IN:=校二浓度:VD104, ENO=>power, OUT=>VD620]  c10 ->
// row 9: c1 ^v  c3 [box]  c6 [box]  c9 [box]
// row 10: c1 ^v  c2 --  c3 [I_DI EN:=power@row10, IN:=标2次数:VW330, ENO=>power, OUT=>VD652]  c4 --  c5 --  c6 [DI_R EN:=power@row10, IN:=VD652, ENO=>power, OUT=>VD652]  c7 --  c8 --  c9 [DIV_R EN:=power@row10, IN1:=平均A2:VD648, IN2:=VD652, ENO=>power, OUT=>平均A2:VD648]  c10 ->
// row 11: c1 ^v  c3 [box]  c6 [box]  c9 [box]
// row 12: c1 ^v  c2 --  c3 [MOV_R EN:=power@row12, IN:=平均A0:VD640, ENO=>power, OUT=>校一a:V2.4]  c4 --  c5 --  c6 [MOV_R EN:=power@row12, IN:=平均A2:VD648, ENO=>power, OUT=>校二a:V2.5]  c7 ->
// row 13: c1 ^v  c3 [box]  c6 [box]
// row 14: c1 ^v  c2 --  c3 [计算KB EN:=power@row14, A1:=校一a:V2.4, 浓度1:=VD608, A2:=校二a:V2.5, 浓度2:=VD620, K=>K:VD158, b=>B:VD162]
// row 15: c1 ^v  c3 [box]
// row 16: c1 ^v  c3 [box]
// row 17: c1 ^v  c2 --  c3 [BLKMOV_W EN:=power@row17, IN:=VW460, N:=5, ENO=>power, OUT=>标定时刻:VW148]  c4 ->
// row 18: c1 ^v  c3 [box]
// row 19: c1 ^v  c2 --  c3 [数据库 EN:=power@row19]
// row 20: c1 ^v  c2 --  c3 [MOV_B EN:=power@row20, IN:=VB93, ENO=>power, OUT=>档位:VB90]  c4 ->
// row 21: c1 ^v  c3 [box]
// row 22: c1 ^  c2 -(S) V20.7, 1
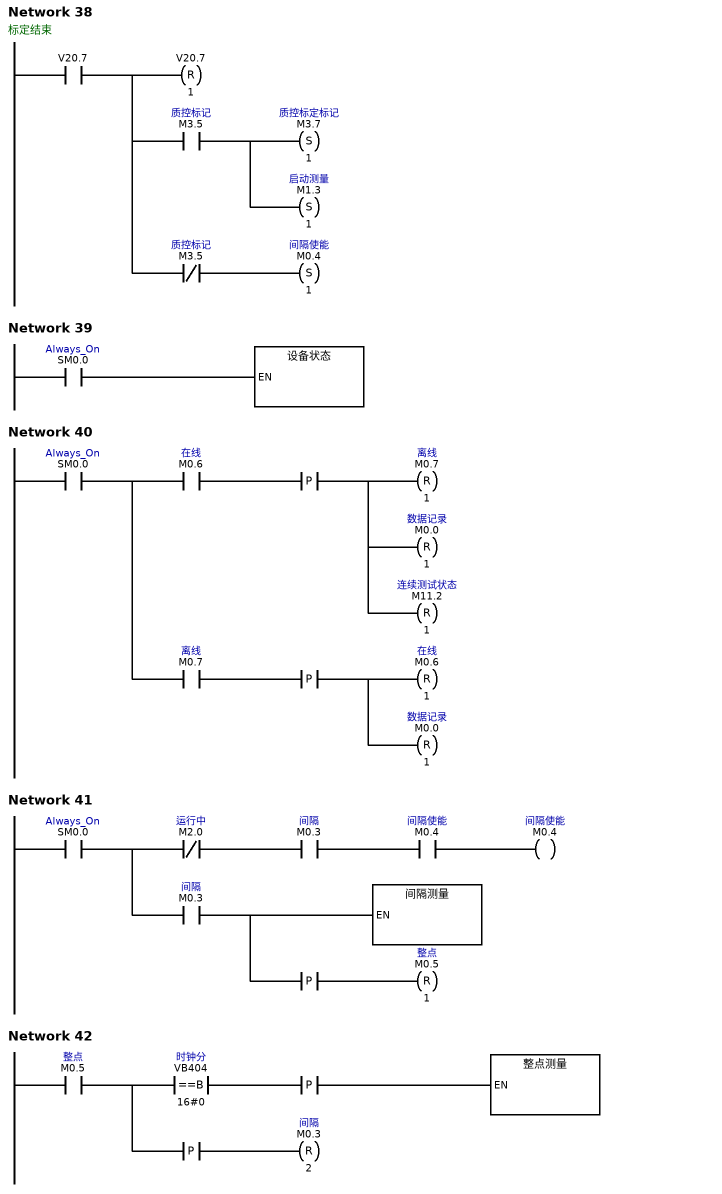
Network 38
// 标定结束
LD     V20.7
LPS
R      V20.7, 1
A      质控标记:M3.5
S      质控标定标记:M3.7, 1
S      启动测量:M1.3, 1
LPP
AN     质控标记:M3.5
S      间隔使能:M0.4, 1
Network 39
LD     Always_On:SM0.0
CALL   设备状态:SBR25
Network 40
LD     Always_On:SM0.0
LPS
A      在线:M0.6
EU
R      离线:M0.7, 1
R      数据记录:M0.0, 1
R      连续测试状态:M11.2, 1
LPP
A      离线:M0.7
EU
R      在线:M0.6, 1
R      数据记录:M0.0, 1
Network 41
LD     Always_On:SM0.0
LPS
AN     运行中:M2.0
A      间隔:M0.3
A      间隔使能:M0.4
=      间隔使能:M0.4
LPP
A      间隔:M0.3
CALL   间隔测量:SBR12
EU
R      整点:M0.5, 1
Network 42
LD     整点:M0.5
LPS
AB=    时钟分:VB404, 16#0
EU
CALL   整点测量:SBR13
LPP
EU
R      间隔:M0.3, 2
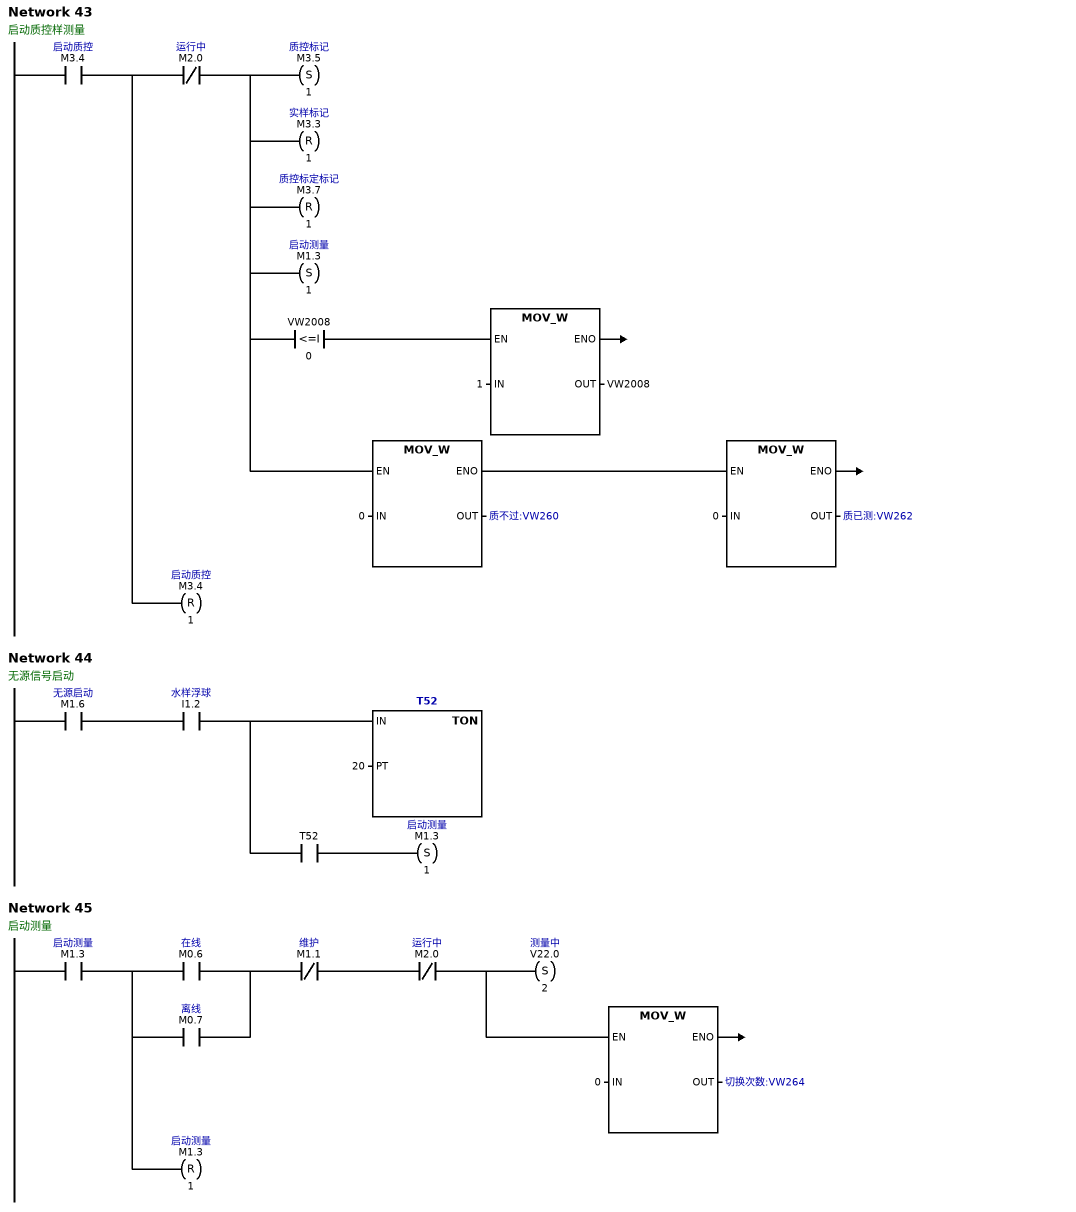
Network 43
// 启动质控样测量
LD     启动质控:M3.4
LPS
AN     运行中:M2.0
LPS
S      质控标记:M3.5, 1
R      实样标记:M3.3, 1
R      质控标定标记:M3.7, 1
S      启动测量:M1.3, 1
AW<=   VW2008, 0
MOVW   1, VW2008
LPP
MOVW   0, 质不过:VW260
AENO
MOVW   0, 质已测:VW262
LPP
R      启动质控:M3.4, 1
Network 44
// 无源信号启动
LD     无源启动:M1.6
A      水样浮球:I1.2
TON    T52, 20
A      T52
S      启动测量:M1.3, 1
Network 45
// 启动测量
LD     启动测量:M1.3
LPS
LD     在线:M0.6
O      离线:M0.7
AN     维护:M1.1
AN     运行中:M2.0
ALD
S      测量中:V22.0, 2
MOVW   0, 切换次数:VW264
LPP
R      启动测量:M1.3, 1
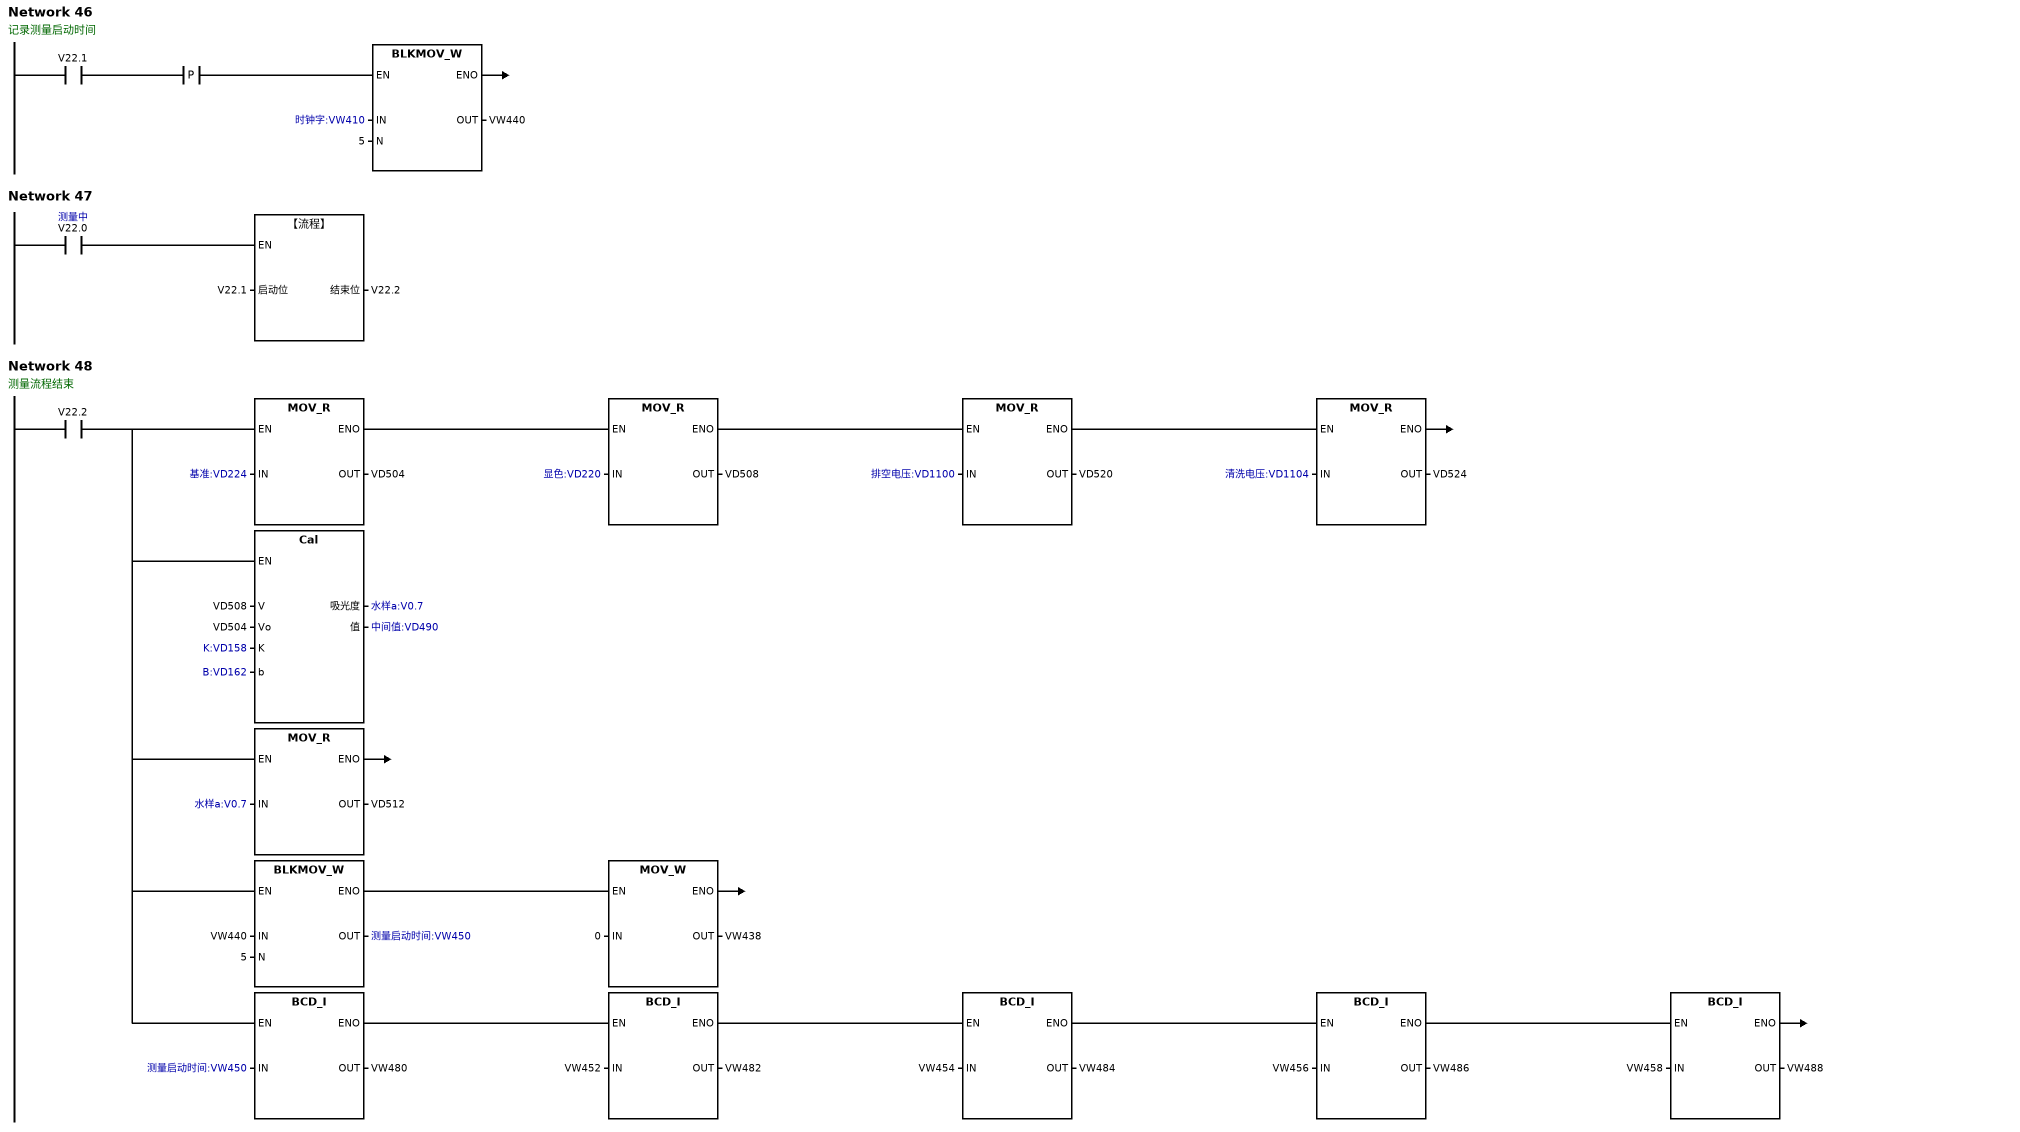
Network 46
// 记录测量启动时间
LD     V22.1
EU
BMW    时钟字:VW410, VW440, 5
Network 47
LD     测量中:V22.0
CALL   【流程】:SBR7, V22.1, V22.2
Network 48
// 测量流程结束
// (network saved uncompiled; LAD cells follow)
// row 0: c0 -| |- V22.2 v  c1 --  c2 [MOV_R EN:=power@row0, IN:=基准:VD224, ENO=>power, OUT=>VD504]  c3 --  c4 --  c5 [MOV_R EN:=power@row0, IN:=显色:VD220, ENO=>power, OUT=>VD508]  c6 --  c7 --  c8 [MOV_R EN:=power@row0, IN:=排空电压:VD1100, ENO=>power, OUT=>VD520]  c9 --  c10 --  c11 [MOV_R EN:=power@row0, IN:=清洗电压:VD1104, ENO=>power, OUT=>VD524]  c12 ->
// row 1: c0 ^v  c2 [box]  c5 [box]  c8 [box]  c11 [box]
// row 2: c0 ^v  c1 --  c2 [Cal EN:=power@row2, V:=VD508, Vo:=VD504, K:=K:VD158, b:=B:VD162, 吸光度=>水样a:V0.7, 值=>中间值:VD490]
// row 3: c0 ^v  c2 [box]
// row 4: c0 ^v  c2 [box]
// row 5: c0 ^v  c1 --  c2 [MOV_R EN:=power@row5, IN:=水样a:V0.7, ENO=>power, OUT=>VD512]  c3 ->
// row 6: c0 ^v  c2 [box]
// row 7: c0 ^v  c1 --  c2 [BLKMOV_W EN:=power@row7, IN:=VW440, N:=5, ENO=>power, OUT=>测量启动时间:VW450]  c3 --  c4 --  c5 [MOV_W EN:=power@row7, IN:=0, ENO=>power, OUT=>VW438]  c6 ->
// row 8: c0 ^v  c2 [box]  c5 [box]
// row 9: c0 ^  c1 --  c2 [BCD_I EN:=power@row9, IN:=测量启动时间:VW450, ENO=>power, OUT=>VW480]  c3 --  c4 --  c5 [BCD_I EN:=power@row9, IN:=VW452, ENO=>power, OUT=>VW482]  c6 --  c7 --  c8 [BCD_I EN:=power@row9, IN:=VW454, ENO=>power, OUT=>VW484]  c9 --  c10 --  c11 [BCD_I EN:=power@row9, IN:=VW456, ENO=>power, OUT=>VW486]  c12 --  c13 --  c14 [BCD_I EN:=power@row9, IN:=VW458, ENO=>power, OUT=>VW488]  c15 ->
// row 10: c2 [box]  c5 [box]  c8 [box]  c11 [box]  c14 [box]
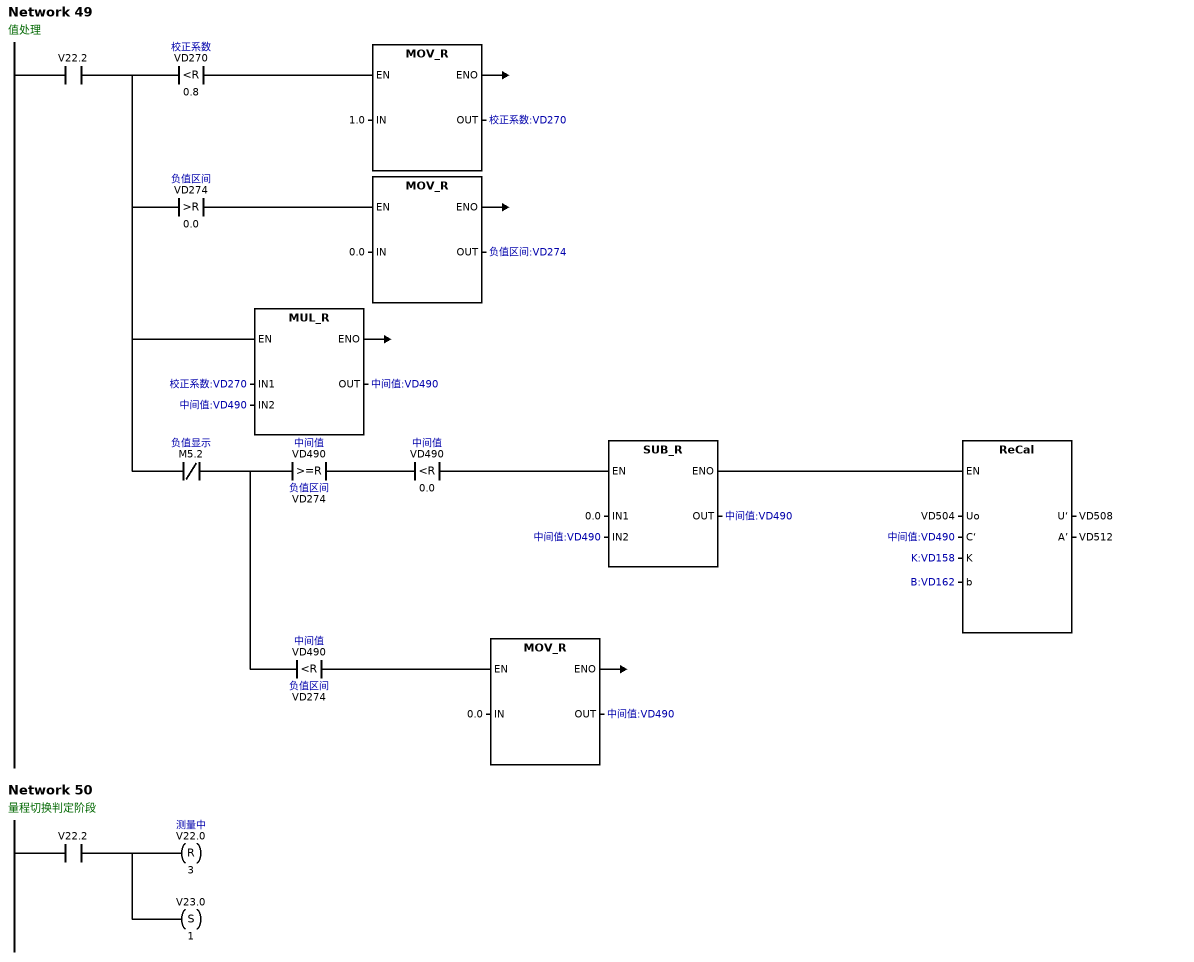
Network 49
// 值处理
LD     V22.2
LPS
AR<    校正系数:VD270, 0.8
MOVR   1.0, 校正系数:VD270
LRD
AR>    负值区间:VD274, 0.0
MOVR   0.0, 负值区间:VD274
LRD
*R     校正系数:VD270, 中间值:VD490
LPP
AN     负值显示:M5.2
LPS
AR>=   中间值:VD490, 负值区间:VD274
AR<    中间值:VD490, 0.0
*R     -1.0, 中间值:VD490
AENO
+R     0.0, 中间值:VD490
AENO
CALL   ReCal:SBR22, VD504, 中间值:VD490, K:VD158, B:VD162, VD508, VD512
LPP
AR<    中间值:VD490, 负值区间:VD274
MOVR   0.0, 中间值:VD490
Network 50
// 量程切换判定阶段
LD     V22.2
R      测量中:V22.0, 3
S      V23.0, 1
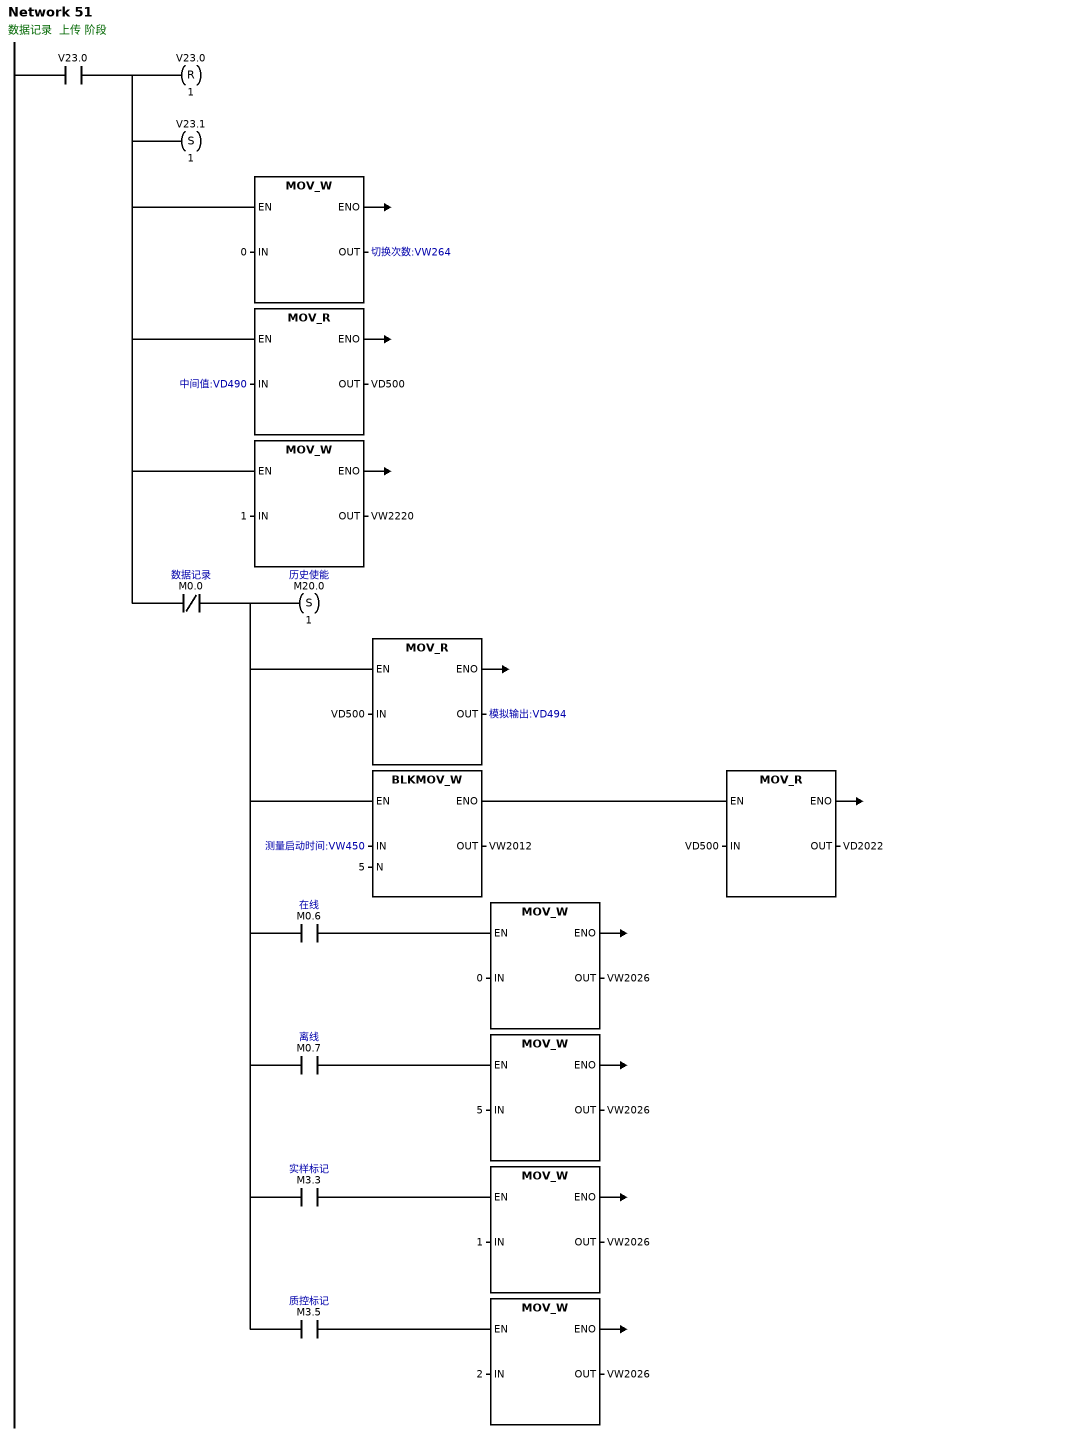
Network 51
// 数据记录  上传 阶段
LD     V23.0
R      V23.0, 1
S      V23.1, 1
MOVW   0, 切换次数:VW264
MOVR   中间值:VD490, VD500
MOVW   1, VW2220
AN     数据记录:M0.0
LPS
S      历史使能:M20.0, 1
MOVR   VD500, 模拟输出:VD494
BMW    测量启动时间:VW450, VW2012, 5
AENO
MOVR   VD500, VD2022
LRD
A      在线:M0.6
MOVW   0, VW2026
LRD
A      离线:M0.7
MOVW   5, VW2026
LRD
A      实样标记:M3.3
MOVW   1, VW2026
LPP
A      质控标记:M3.5
MOVW   2, VW2026
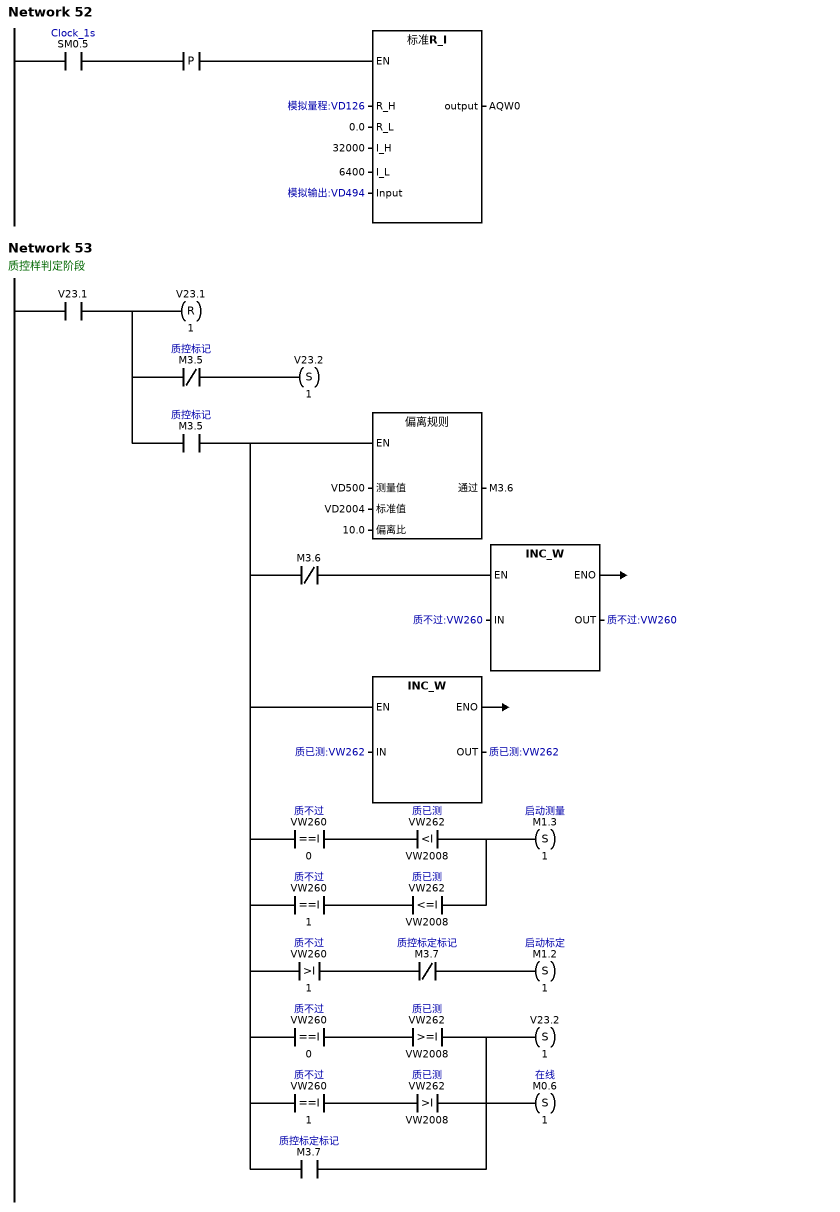
Network 52
LD     Clock_1s:SM0.5
EU
CALL   标准R_I:SBR23, 模拟量程:VD126, 0.0, 32000, 6400, 模拟输出:VD494, AQW0
Network 53
// 质控样判定阶段
LD     V23.1
LPS
R      V23.1, 1
AN     质控标记:M3.5
S      V23.2, 1
LPP
A      质控标记:M3.5
LPS
CALL   偏离规则:SBR16, VD500, VD2004, 10.0, M3.6
AN     M3.6
INCW   质不过:VW260
LRD
INCW   质已测:VW262
LRD
LDW=   质不过:VW260, 0
AW<    质已测:VW262, VW2008
LDW=   质不过:VW260, 1
AW<=   质已测:VW262, VW2008
OLD
ALD
S      启动测量:M1.3, 1
LRD
AW>    质不过:VW260, 1
AN     质控标定标记:M3.7
S      启动标定:M1.2, 1
LPP
LDW=   质不过:VW260, 0
AW>=   质已测:VW262, VW2008
LDW=   质不过:VW260, 1
AW>    质已测:VW262, VW2008
OLD
O      质控标定标记:M3.7
ALD
S      V23.2, 1
S      在线:M0.6, 1
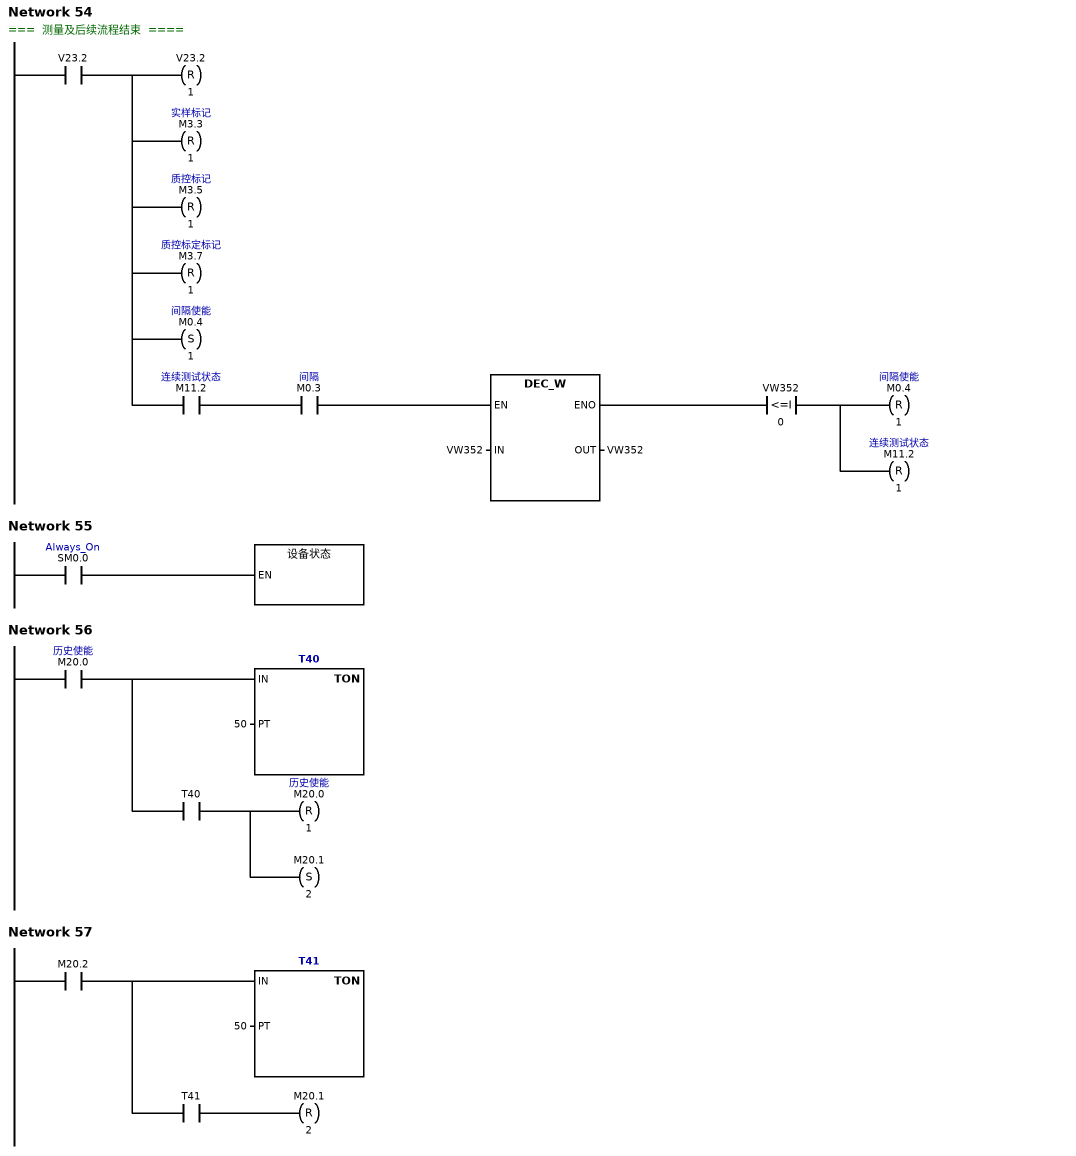
Network 54
// ===  测量及后续流程结束  ====
LD     V23.2
R      V23.2, 1
R      实样标记:M3.3, 1
R      质控标记:M3.5, 1
R      质控标定标记:M3.7, 1
S      间隔使能:M0.4, 1
A      连续测试状态:M11.2
A      间隔:M0.3
DECW   VW352
AENO
AW<=   VW352, 0
R      间隔使能:M0.4, 1
R      连续测试状态:M11.2, 1
Network 55
LD     Always_On:SM0.0
CALL   设备状态:SBR25
Network 56
LD     历史使能:M20.0
TON    T40, 50
A      T40
R      历史使能:M20.0, 1
S      M20.1, 2
Network 57
LD     M20.2
TON    T41, 50
A      T41
R      M20.1, 2
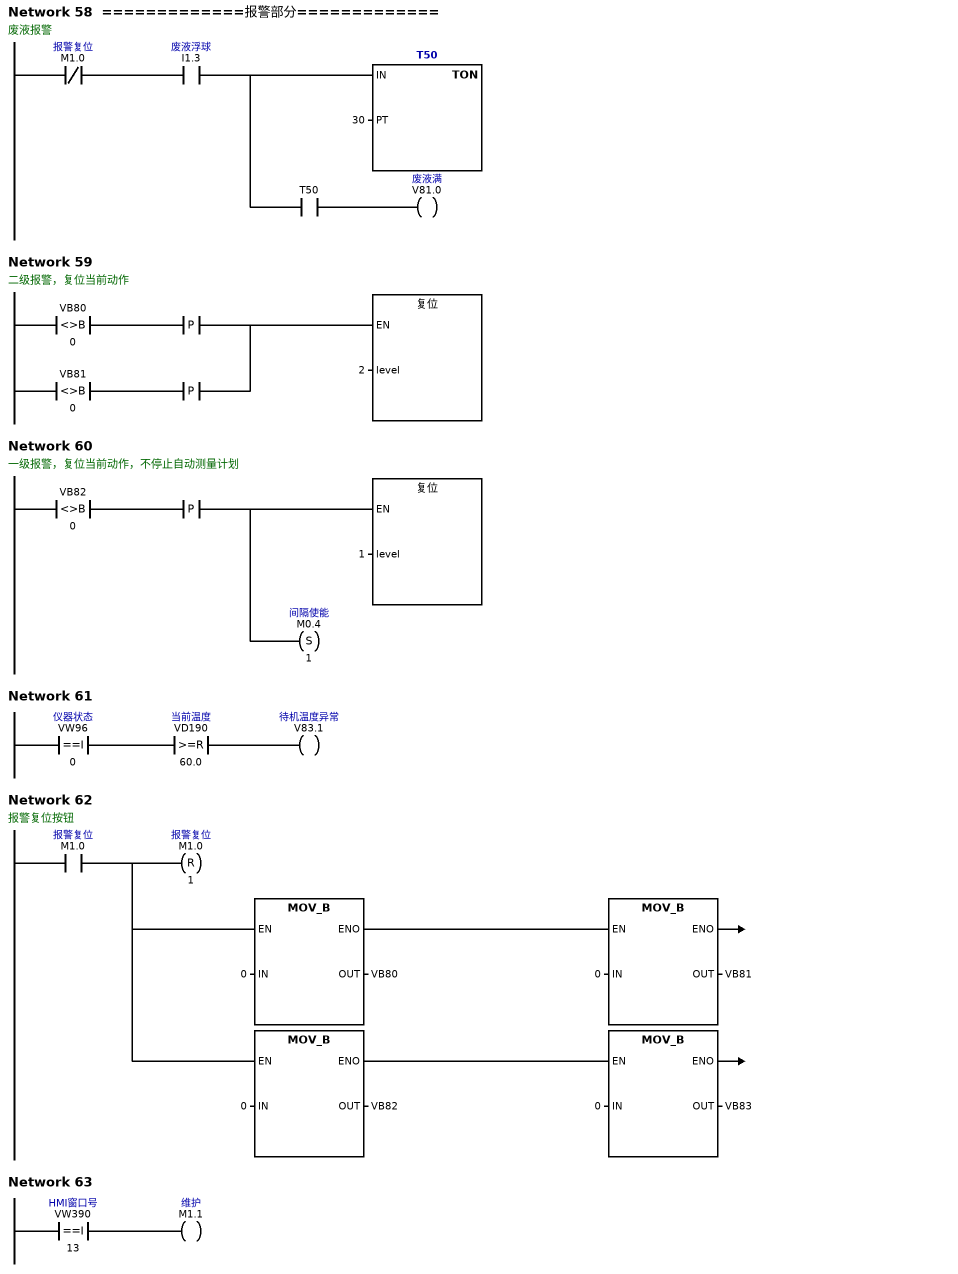
Network 58 // =============报警部分=============
// 废液报警
LDN    报警复位:M1.0
A      废液浮球:I1.3
TON    T50, 30
A      T50
=      废液满:V81.0
Network 59
// 二级报警，复位当前动作
LDB<>  VB80, 0
EU
LDB<>  VB81, 0
EU
OLD
CALL   复位:SBR34, 2
Network 60
// 一级报警，复位当前动作，不停止自动测量计划
LDB<>  VB82, 0
EU
CALL   复位:SBR34, 1
S      间隔使能:M0.4, 1
Network 61
LDW=   仪器状态:VW96, 0
AR>=   当前温度:VD190, 60.0
=      待机温度异常:V83.1
Network 62
// 报警复位按钮
LD     报警复位:M1.0
LPS
R      报警复位:M1.0, 1
MOVB   0, VB80
AENO
MOVB   0, VB81
LPP
MOVB   0, VB82
AENO
MOVB   0, VB83
Network 63
LDW=   HMI窗口号:VW390, 13
=      维护:M1.1
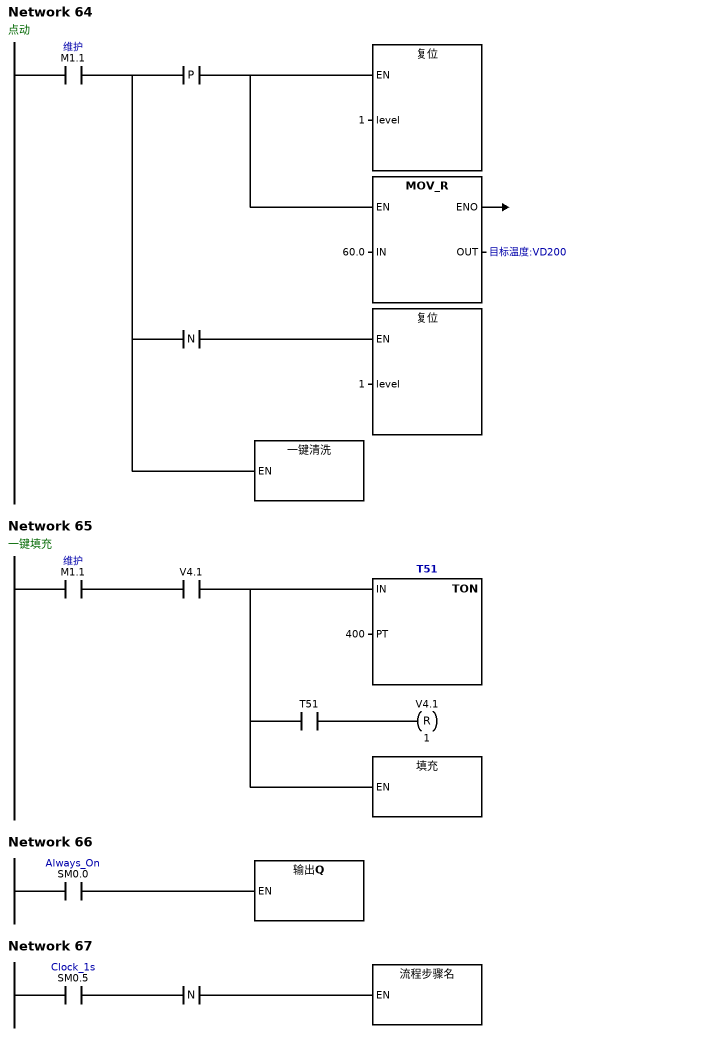
Network 64
// 点动
LD     维护:M1.1
LPS
EU
CALL   复位:SBR34, 1
MOVR   60.0, 目标温度:VD200
LPP
LPS
ED
CALL   复位:SBR34, 1
LPP
CALL   一键清洗:SBR40
Network 65
// 一键填充
LD     维护:M1.1
A      V4.1
LPS
TON    T51, 400
A      T51
R      V4.1, 1
LPP
CALL   填充:SBR39
Network 66
LD     Always_On:SM0.0
CALL   输出Q:SBR8
Network 67
LD     Clock_1s:SM0.5
ED
CALL   流程步骤名:SBR35
